(* CODESYS project IndraLogic.project

Project tree, tasks and I/O mapping:
  IndraMotionMlc1 : IndraMotion MLC L75, Bosch Rexroth AG, order no. R911173004, version 14.22.170.0
    application Application
      libraries: SysCallback23, * (System); Util, * (System); RIL_SocketComm, * (System); SysTime23, * (System); SysTaskInfo23, * (System); RIL_CheckRtv, * (System); ML_TechMotion, * (System); SysSocket23, * (System); SysTime, 3.4.1.20 (System); ML_TechInterface, 14.20.30.0 (System); ML_TechBase, 14.18.0.0 (System); VisuDialogs, * (System); ML_TechMotionBase, * (System); RIL_LoopControl, 14.22.36.0 (System); RIL_OpcUaServer, * (System); RIL_OpcUaClient, * (System); IoDrvModbusTCP, * (3S - Smart Software Solutions GmbH)
      task motion (externalevent, external event EVENT_OP_MODE_MOTION_CYCLIC, priority 2) calls P_Position_and_MJD [add POU_1MS below for frequency response tests], P_EL_VEL_MODE, P_PID_antibacklash, P_UDP_To_NTP, POU_20200525, P_Track_cubic, P_Simulation [Just for Simulation PLC remove for pedestal deploy]
      task panel (cyclic, interval t#20ms, priority 7) calls P_remote_local, P_power_on_Sim, P_power_off_TCP
      task TCP (cyclic, interval 10 ms, priority 4) calls P_Opcua_Azimuth [Removed P_TCP_with_SCC], P_Opcua_Elevation, P_Opcua_FeedIndexer, P_Opcua_Safety, P_Opcua_CommandArbiter, P_Opcua_Time_cds, P_Opcua_Management, P_UDP_with_DAM, P_Opcua_Tracking, P_Opcua_Pointing
      task other (cyclic, interval 100 ms, priority 8) calls Test_move, PlcProg
      task AutoStow (cyclic, interval 60000 ms, priority 20) calls P_AutoStow
      function CheckBounds [ST]
      Symbols
      global variables MlcVarGlobal
      POUs/
        Motion/
          program P_PID_antibacklash [ST]: A_PID
          program P_power_off_TCP [LD]
          program P_power_on_TCP [LD]
          program Test_move [ST]: power_move
          program POU_20200525 [ST]
          program PlcProg [ST]
          program P_Position_and_MJD [ST]: A_Write_Limit_Value
          program P_EL_VEL_MODE [ST]
          program P_Track_cubic [ST]: A_track_fuction_blocks, A_StaticPM, A_DynamicPM, A_AmbTempPM, A_Sim_track_function_blocks
          program POU_1MS [ST]: P_Move
          program P_power_on_Sim [LD]
          program P_Read_Parameters [ST]: A_Read_Parameter
          program P_interpolator [ST]: A_track_fuction_blocks, A_StaticPM, A_DynamicPM, A_AmbTempPM, A_Sim_track_function_blocks
        Panel Function/
          program P_LED [ST]: A_w_P304
          program P_Lock_Panel_TCP [ST]: A_LOCK
          program P_Panel_Jog [ST]: A_axes_running
          program P_read_drv_IO [LD]
          program P_remote_local [ST]: A_clear_error
        TCP/
          Message/
            function block FB_add_vector_old_mode [ST]
            function block FB_MSG [ST]
            function block FB_Str_Divide [ST]
            function F_I_number [ST]
            function F_reduce_to_1_bit [ST]
            function F_reduce_to_4_bit [ST]
            function F_RPL [ST]
            function F_RPL_1 [ST]
            function F_RPL_2 [ST]
            function F_Trim [ST]
            function deg2rad [ST]
            function Encoder_to_motor [ST]
            function block FB_add_vector [ST]
            function Encoder_to_motor_old [ST]
            function P_CLOSE_LOOP [ST]
            function block FB_Caculate_position_1 [ST]
            function F_cyclic_position [ST]
            function block CRC16_MODBUS [ST]
          program P_GSTAT_K2STAT [ST]: A_Read_Parameter
          program P_TCP_with_SCC [ST]: Async_TCP, A_RECV, A_SCC_GOTO, A_SCC_POWER, A_SCC_STOP, A_SEND
          program P_UDP_with_DAM [ST]: Async_TCP, A_RECV, A_SEND
        Time Control/
          function F_NTP_Head [ST]
          program P_UDP_To_NTP [ST]: A_NTP_to_Master, A_UDP
        program Annotation [ST]
        Useless/
          program MotionProg [ST]: P_MOTION
          program POU_1MS_Az_freq [ST]
          program POU_1MS_old_mode [ST]: P_Move
        OPCUA/
          OPCUA_Node/
            program P_Opcua_Azimuth [ST]
            program P_Opcua_Elevation [ST]
            program P_Opcua_FeedIndexer [ST]
            program P_Opcua_Safety [ST]: A_STOW, A_Interlock_Estop
            program P_Opcua_CommandArbiter [ST]
            program P_Opcua_Time_cds [ST]: Get_Time
            program P_Opcua_Management [ST]: A_STOP, A_GOTO, A_CLR_ERR
            program P_Opcua_Pointing [ST]: A_Utils
            program P_Opcua_Tracking [ST]: A_Utils
          OPCUA_Method/
            function block fb_Axis [ST]
            function block fb_CommandArbiter [ST]
            function block fb_Management [ST]
            function block fb_Pointing [ST]
            function block fb_Safety [ST]
            function block fb_Time_cds [ST]
            function block fb_Tracking [ST]
            function block fb_Time_Commands [ST]: SetTimeSource
            function block fb_Pointing_Commands [ST]: AmbTempCorrSetup, PmCorrOnOff, StaticPmSetup, TiltCalSetup
            function block fb_Tracking_Commands [ST]: TrackLoadStaticOff, TrackLoadTable, TrackStart, TrackStartPoly
            function block fb_Mngmt_Commands [ST]: Activate, DeActivate, Move2Band, Reset, SetOnSourceThreshold, SetPowerMode, Slew2AbsSingleAx, Slew2AbsAzEl, Slew2RelSingleAx, Slew2RelAzEl, Stop, Stow, TrackStartDM, TrackStartPolyDM
            function block fb_CommandArbiter_Commands [ST]: TakeAuth, ReleaseAuth, Get_Time
            function block fb_Safety_Commands [ST]: InterlockAck, MoveStowPin
        Simulation/
          program P_Simulation [ST]
        AutoStow/
          program P_AutoStow [ST]
      global variables Global_Variables
      Data types/
        data type Stack_buffer
        data type UDP_PACKET
        data type Angle_Mark
        data type ANG_MARK
      global variables UserConstGlobal
      global variables UserVarGlobal
      AxisInterface/
        Documentation/
        Type/
          data type TE_PLC_CYCLES_TIME
          Control/
            data type TE_AXIS_ADMINISTRATION
            data type TE_AXIS_CONTROL_TYPE01
            data type TE_AXIS_POSITIONING
            data type TE_AXIS_SETUP_MODE
            data type TE_AXIS_SYNCHRONISATION
            data type TE_AXIS_TORQUE
            data type TE_AXIS_VELOCITY
          Status/
            data type TE_AXIS_ADMIN_STATUS
            data type TE_AXIS_DATA_STATUS
            data type TE_AXIS_DIAGNOSIS
            data type TE_AXIS_POS_STATUS
            data type TE_AXIS_SETUP_MODE_STATUS
            data type TE_AXIS_STATUS_TYPE01
            data type TE_AXIS_SYNC_STATUS
            data type TE_AXIS_VEL_STATUS
        Visualizations/
          AxisModes/
            text list AxisMode
            text list ExecutionMode
            text list ProfileEntry
            text list StartMode
            text list SyncDirection
            text list SyncType
            visualisation Axis_Overview
            visualisation Position_mode
            visualisation Profile_mode
            visualisation Synchronization_mode
            visualisation Torque_mode
            visualisation Velocity_mode
          ImcInterface/
            text list ImcModeControl
            text list ImcModeStatus
            visualisation ImcControl
            visualisation ImcInterface_Status_Control
            visualisation ImcStatus
          SystemOverview/
            text list ErrorIDCode
            text list ErrorTable
            visualisation System_Overview
            visualisation System_Overview_All_Axis
            visualisation System_Overview_header
          Utilities/
            visualisation AdjustPosition
            visualisation AdjustVelocity
        global variables Global_AxIf_Const
        global variables Global_Axis_Interface
        function block TE_AxisInitAllAxisType01 [ST]
        function block TE_AxisInterface [ST]: actAngleOffset, actCopyAxisData_HMI, actPhaseShift, actPMSpecialErrors, actRetriggerOpMode, actSetupMode, actSyncAccVel, mClearError, mGetOpMode, mInitExtension, mSetOpMode
        program TE_AxisInterfaceType01Prog [ST]: actInitWarmStart
        program _Readme [ST]
      trace/
        trace Trace_simulation (task motion): r_write_position_az, r_write_position_el
        trace Trace_1 (task motion): r_pos_az, r_torque_1, r_torque_2, Global_Variables.i_speed_1, Global_Variables.i_speed_2, i_pos_cmd_1
        trace Trace_2 (task motion, trigger Positive on POU_1MS.r_new_cmd_pos): P_Position_and_MJD.r_test_value, r_following_3, P_Position_and_MJD.b_sign_delay, P_Position_and_MJD.test_1, r_compensation_abs, AxisData[3].rActualTorqueForce_i, r_track_error[2], ML_Base.AxisData[11].rActualPosition_i, r_pos_motor3, P_track_cubic.r_write_position_el, r_vel_EL, P_Track_cubic.r_following_31, P_Position_and_MJD.r_source_to_elevation
        trace Trace_EL_freq_res (task motion): r_pos_motor3, ML_Base.AxisData[11].rActualPosition_i, POU_1MS.Frequency_vel, POU_1MS.vel_freq, POU_1MS.T_period, AxisData[3].rActualVelocity_i, AxisData[3].rActualTorqueForce_i, POU_1MS.torque_freq, Pos_EL_Aim, arAxisCtrl_gb[Drive3.AxisNo].VelMode.Velocity
        trace Trace_compensation (task motion, trigger Positive on POU_1MS.r_new_cmd_pos): r_pos_motor3, ML_Base.AxisData[11].rActualPosition_i, P_Position_and_MJD.test_1, r_track_error[2], AxisData[3].rActualTorqueForce_i, P_Track_cubic.r_write_position_el, P_Track_cubic.r_offset_t, P_Track_cubic.r_test_offset_az, P_Track_cubic.r_test_offset_el
        trace Trace_random_array (task track_task, trigger Positive on POU_1MS.r_new_cmd_pos): ML_Base.AxisData[11].rActualPosition_i, r_pos_motor3, POU_1MS.vel_random_array, AxisData[3].rActualVelocity_i, AxisData[3].rActualTorqueForce_i, POU_1MS.i_test_count, POU_1MS.i_random_count, POU_1MS.vel_freq
        trace Trace_random_array_AZ (task track_task, trigger Positive on POU_1MS.r_new_cmd_pos): ML_Base.AxisData[1].rActualPosition_i, axisdata[1].rActualPosition_i, axisdata[2].rActualPosition_i, POU_1MS.vel_random_array, AxisData[1].rActualVelocity_i, AxisData[1].rActualTorqueForce_i, AxisData[2].rActualTorqueForce_i, POU_1MS.i_test_count, POU_1MS.i_random_count, POU_1MS.vel_random_array
        trace Trace_AZ_freq_res (task motion): ML_Base.AxisData[1].rActualPosition_i, axisdata[1].rActualPosition_i, axisdata[2].rActualPosition_i, POU_1MS.Frequency_vel, AxisData[1].rActualVelocity_i, AxisData[2].rActualVelocity_i, AxisData[1].rActualTorqueForce_i, AxisData[2].rActualTorqueForce_i, POU_1MS.torque_freq, ML_Base.AxisData[11].rActualPosition_i, r_following_1, r_following_3
        trace Trace_EL_VEL_MODE (task motion): r_pos_el, Pos_EL_error, AxisData[3].rActualTorqueForce_i, Pos_EL_Aim, b_step_running, r_vel_EL, AxisData[3].rActualVelocity_i
      global variables PLC_PRG
      OPC_UA_Symbols_Objects/
        data type AxisSelectType
        data type AxisStateType
        data type BandType
        data type CmdResponseType
        data type DscCmdAuthorityType
        data type DscStateType
        data type DscTimeSyncSourceType
        data type InterpolType
        data type LoadModeType
        data type SafetyStateType
        data type StowPinStatusType
        data type TimeSourceType
        data type TiltOnType
      OPCUA_Data_type/
        data type AmbTempParam_Type
        data type AxisErrorStatus_Type
        data type MngmtStatus_Type
        data type MotorStatus_Type
        data type StaticPmParam
        data type TableStatus_type
        data type TiltmeterParam
        data type TiltmeterSubParam
        data type MngmtWarningStatus_Type
        data type SafetyStatus_Type
        data type Time_cdsStatus_type
        data type PointingStatus_Type
        data type TrackingStatus_Type
        data type PolyStatus_type
        data type PowerStatus_Type
        data type AxisWarning_Type
        data type MngmtErrorStatus_Type
        data type TempHumidStatus_Type
        data type NamePlate_Type
        data type CommandArbiter_Status_Type
        data type AxisGeneralStatus_Type
      trace Azimuth_Desired (task TCP, trigger Positive on b_track_on): Tracking.Status.p_desired_Az, Tracking.Status.p_desired_El
    Onboard_I_O : Onboard I/O, Bosch Rexroth AG, version 13.6.2.0
        unmapped channels: OnboardIn, OnboardOut
    Inline_I_O : Inline I/O, Bosch Rexroth AG, version 12.8.2.0
      R_IB_IL_24_DI_32_HD : R-IB IL 24 DI 32/HD, Bosch Rexroth AG, order no. R911170753, R911297188, version 0.0.0.1
          unmapped channels: Input0
      R_IB_IL_24_DO_32_HD : R-IB IL 24 DO 32/HD, Bosch Rexroth AG, order no. R911170411, R911297191, version 0.0.0.1
          unmapped channels: Output0
    Not_Used : Not Used, Bosch Rexroth AG, version 12.2.0.0
    EtherNet_IP_Adapter : EtherNet/IP Adapter, Bosch Rexroth AG, version 14.22.10.0
    Sercos_III_Master : SercosIII Master, Rexroth, order no. 1, version 14.6.0.0
    EtherNet_IP_Adapter_on_Eng_Port : EtherNet/IP Adapter on Eng.-Port, Bosch Rexroth AG, version 12.10.2.0
      _8_Byte_Input : 8 Byte Input, Bosch Rexroth AG, version 12.10.2.0
          unmapped channels: Channel1
      _8_Byte_Output_4Byte_Run_Header : 8 Byte Output + 4Byte Run Header, Bosch Rexroth AG, version 12.10.2.0
          unmapped channels: Channel1
  libraries: Time and Date, 3.5.7.0 (3S - Smart Software Solutions GmbH); Util, * (System); RIL_OpcUaServer, 14.22.0.1 (System); RIL_LoopControl, 14.22.36.0 (System); RIL_EtherNetIPAdapter, 14.4.0.0 (System); ML_PLCopen, 14.22.32.0 (System); IoDrvModbusTCP, * (3S - Smart Software Solutions GmbH)
  text list GlobalTextList
  visualisation Visualization
*)

// IndraMotionMlc1/Application/OPCUA_Data_type/AmbTempParam_Type
TYPE AmbTempParam_Type :
STRUCT
	AmbTempParam1:LREAL;
	AmbTempParam2:LREAL;
	AmbTempParam3:LREAL;
	AmbTempParam4:LREAL;
	AmbTempParam5:LREAL;
	AmbTempParam6:LREAL;
	Filt_dt:LREAL;
END_STRUCT
END_TYPE

// IndraMotionMlc1/Application/Data types/Stack_buffer
(*construction of stack *)
TYPE Stack_buffer :
STRUCT
	TAIoffset:LREAL;
	Azimuth:LREAL;
	Elevation:LREAL;
	//FeedIndexer:LREAL;
	//Elevation_ori:LREAL;
END_STRUCT
END_TYPE

// IndraMotionMlc1/Application/Data types/UDP_PACKET
TYPE UDP_PACKET :(*constrution of NTP header*)
STRUCT
	(*NTP packet = NTP header 16bytes + Four TimeStamps 32 byte = 48byte*)
	NTP_Header :ARRAY[1..4] OF BYTE;
	NTP_Root_Delay:ARRAY[1..4] OF BYTE;
	NTP_Root_Dispersion:ARRAY[1..4] OF BYTE;
	NTP_Reference_Identifier:ARRAY[1..4] OF BYTE;

	NTP_Reference_Timestamp:ARRAY[1..2] OF DWORD;
	NTP_Originate_Timestamp:ARRAY[1..2] OF DWORD;
	NTP_Receive_Timestamp:ARRAY[1..2] OF DWORD;
	NTP_Transmit_Timestamp:ARRAY[1..2] OF DWORD;
END_STRUCT
END_TYPE

// IndraMotionMlc1/Application/Data types/Angle_Mark
TYPE Angle_Mark :
STRUCT
	stui_RSV : DINT;			//补齐8字节，对齐地址
	stui_SID : DINT;
	stui_DID : DINT;
	stui_BID : DINT;
	stui_DataLen : DINT;
	sti_Year : DINT;
	sti_Month : DINT;
	sti_Day : DINT;
	sti_Hour : DINT;
	sti_Minute : DINT;
	sti_Second : DINT;
	sti_MilSecond : DINT;
	std_GEOAngle_AZ : LREAL;
	std_GEOAngle_EL : LREAL;
END_STRUCT
END_TYPE

// IndraMotionMlc1/Application/Data types/ANG_MARK
TYPE ANG_MARK :
UNION
	st_ANGMARK : Angle_Mark;
	ANG_SEND : ARRAY [1..64] OF BYTE;
END_UNION
END_TYPE

// IndraMotionMlc1/Application/AxisInterface/Type/TE_PLC_CYCLES_TIME
TYPE TE_PLC_CYCLES_TIME :
STRUCT

     udiMinimumTime  : UDINT  := 1000000;
     udiActualTime   : UDINT  := 0;
     udiMaximumTime  : UDINT  := 0;

END_STRUCT
END_TYPE

// IndraMotionMlc1/Application/AxisInterface/Type/Control/TE_AXIS_ADMINISTRATION
// Online changes in declaration of axis-interface need too much time -> not allowed because risk of F5180006 
// InhibitOnlineChange = 0x1000000 has to be set decimal 16777216
{attribute 'signature_flag' := '16777216'} 
TYPE TE_AXIS_ADMINISTRATION EXTENDS MB_AXIS_ADMINISTRATION:
STRUCT
  (* add your extensions below here |  Erweiterungen hier einfuegen*)

  (* user extensions | Anwender Erweiterungen *)
  
  RetriggerOpMode: BOOL;   // Restart the same OpMode again, e.g. MoveRelative with same distance	

END_STRUCT
END_TYPE

// IndraMotionMlc1/Application/AxisInterface/Type/Control/TE_AXIS_CONTROL_TYPE01
// Online changes in declaration of axis-interface need too much time -> not allowed because risk of F5180006 
// InhibitOnlineChange = 0x1000000 has to be set decimal 16777216
{attribute 'signature_flag' := '16777216'} 
TYPE TE_AXIS_CONTROL_TYPE01:

STRUCT
    Admin:      TE_AXIS_ADMINISTRATION; (* Administration of the axis | Verwaltung der Achse *)

    PosMode:    TE_AXIS_POSITIONING; (* operating mode positioning (absolute, rel. and additive)
      Positionierbetrieb (absolut, relativ und additiv) *)

    VelMode:    TE_AXIS_VELOCITY; (* operating mode velocity control | Geschwindigkeitsregelung *)

    SyncMode:   TE_AXIS_SYNCHRONISATION; (* operating mode synchronisation (phase, vel, and cam)
      Synchronbetriebsarten (Winkelsync., Geschwindigkeitssync. und Kurvenscheibe) *)
			
    TorqueMode: TE_AXIS_TORQUE; (* operating mode torque/force control | Drehmoment-/Kraftregelung *)

    (* add your extensions below here, keep the elements above
       Erweiterungen hier einfuegen, Elemente oberhalb nicht veraendern *)

    (* user extensions | Anwender Erweiterungen *)
    
	  // Jog/Homing functionality | Tipp/Einrichtfunktionen 
    SetupMode:  TE_AXIS_SETUP_MODE; 
	
END_STRUCT

END_TYPE

// IndraMotionMlc1/Application/AxisInterface/Type/Control/TE_AXIS_POSITIONING
    (*************** - setpoints of positioning mode ******************)
    (*************** - Positions-Sollwerte           ******************)
// Online changes in declaration of axis-interface need too much time -> not allowed because risk of F5180006 
// InhibitOnlineChange = 0x1000000 has to be set decimal 16777216
{attribute 'signature_flag' := '16777216'} 
TYPE TE_AXIS_POSITIONING EXTENDS MB_AXIS_POSITIONING:
STRUCT

    (* position for an absolute move (in technical unit[u]) (negative or positive)
      - start moving with "ModePosAbs" (MC_MoveAbsolute)
      Note: cyclic checked AND transmitted on change (EnableCyclicScanning = TRUE) 
      ------------------------------------------------------------------------------
      Zielposition, absolut (Einheit: [u]) (negativ oder positiv)
      - Freigabe mit "ModePosAbs" (MC_MoveAbsolute)
      Hinweis: wird permanent zyklisch verarbeitet (EnableCyclicScanning = TRUE) *)
    // Position:        REAL;

    (* distance for a relative or additive move (in technical unit[u]) (negative or positive)
      - start moving with "ModePosRel" or "ModePosAdd" (MC_MoveRelative, MC_MoveAdditive) 
      Note: cyclic checked AND transmitted on change (EnableCyclicScanning = TRUE) 
      ------------------------------------------------------------------------------
      Relativer / additiver Sollwert (Einheit: [u]) (negativ oder positiv )
      - Freigabe mit "ModePosRel" oder "ModePosAdd" (MC_MoveRelative, MC_MoveAdditive) 
      Hinweis: wird permanent zyklisch verarbeitet (EnableCyclicScanning = TRUE) *)
     // Distance:        REAL;

    (* maximum velocity (always positive) (not necessarily reached) [u/s]
      - start moving with "ModePosAbs" or "ModePosRel" or "ModePosAdd" 
        (MC_MoveAbsolute, MC_MoveRelative, MC_MoveAdditive) 
      Note: cyclic checked AND transmitted on change (EnableCyclicScanning = TRUE) 
      ------------------------------------------------------------------------------
      Positioniergeschwindigkeit , (Einheit: [u/s]) (positiv eingeben)
      - Freigabe mit "ModePosAbs" oder "ModePosRel" oder "ModePosAdd" 
        (MC_MoveAbsolute, MC_MoveRelative, MC_MoveAdditive) 
      Hinweis: wird permanent zyklisch verarbeitet (EnableCyclicScanning = TRUE) *)
    // Velocity:        REAL:=10.0;

    (* Value of the acceleration (always positive) (increasing energy of the motor) [u/s2]
      - start moving with "ModePosAbs" or "ModePosRel" or "ModePosAdd" 
        (MC_MoveAbsolute, MC_MoveRelative, MC_MoveAdditive) 
      ------------------------------------------------------------------------------
      Beschleunigung (Einheit: [u/s2]) (nur positive Werte)             
      - Freigabe mit "ModePosAbs" oder "ModePosRel" oder "ModePosAdd" 
        (MC_MoveAbsolute, MC_MoveRelative, MC_MoveAdditive) *)
    // Acceleration:    REAL:=10.0;

    (* Value of the deceleration (always positive) (decreasing energy of the motor) [u/s2]
      - start moving with ModePosAbs or ModePosRel or ModePosAdd 
        (MC_MoveAbsolute, MC_MoveRelative, MC_MoveAdditive) 
      ------------------------------------------------------------------------------
      Verzoegerung, (Einheit: [u/s2]) (nur positive Werte)            
      - Freigabe mit "ModePosAbs" oder "ModePosRel" oder "ModePosAdd" 
        (MC_MoveAbsolute, MC_MoveRelative, MC_MoveAdditive) *)
    // Deceleration:    REAL:=10.0;
	
(* add your extensions below here, keep the elements above
   Erweiterungen hier einfuegen, Elemente oberhalb nicht veraendern *)

(* user extensions | Anwender Erweiterungen *)

END_STRUCT
END_TYPE

// IndraMotionMlc1/Application/AxisInterface/Type/Control/TE_AXIS_SETUP_MODE
// Online changes in declaration of axis-interface need too much time -> not allowed because risk of F5180006 
// InhibitOnlineChange = 0x1000000 has to be set decimal 16777216
{attribute 'signature_flag' := '16777216'} 
TYPE TE_AXIS_SETUP_MODE :
  STRUCT
    Enable:          BOOL;	  (* Enable setup mode  | Freigabe Einrichtbetrieb
      - activates Power                        | - aktiviert Antriebsfreigabe *)
 
    JogPlus:         BOOL;  	(* Jog +            | Tippen + 
      - activates ModeVelocity with pos. Vel   | - aktiviert ModeVelocity mit pos. Vel *)
 
    JogMinus:        BOOL;    (* Jog -            | Tippen - 
      - activates ModeVelocity with pos. Vel   | - aktiviert ModeVelocity mit neg. Vel *)

    JogPosControl:   BOOL:=FALSE; (* Select jog in velocity or positioning control | Auswahl tippen in Geschwindigkeits- oder Lageregelung 
           TRUE = jog in positioning control | TRUE = tippen in Lageregelung *)

	  (* Homing *)
    {attribute 'analysis' := '-27'} // disable static code analysis rule 27, check of same names 
    Homing: BOOL;  (* - activates ModeHoming|SetAbsRef|ModesPosAbs | activiert ModeHoming|SetAbsRef|ModesPosAbs
        depending on axistype/-configuration       | abhängig vom Achstyp/-konfiguration       *) 

	
    Vel:    REAL:= 10; (* jog/homing velocity  | Tipp-/Referenzfahrgeschwindigkeit *)
	
    Accel:  REAL:= 10; (* jog/homing ac/deceleration  | Tipp/Referenzfahr (brems)beschleunigung *)
  END_STRUCT
END_TYPE

// IndraMotionMlc1/Application/AxisInterface/Type/Control/TE_AXIS_SYNCHRONISATION
    (*************** - setpoint of synchronous motion ******************)
// Online changes in declaration of axis-interface need too much time -> not allowed because risk of F5180006 
// InhibitOnlineChange = 0x1000000 has to be set decimal 16777216
{attribute 'signature_flag' := '16777216'} 
TYPE TE_AXIS_SYNCHRONISATION EXTENDS MB_AXIS_SYNCHRONISATION:
STRUCT

    (* Electronic gear input revolution
      - "ModeSyncPhase", "ModeSyncVel", "ModeSyncCam", "ModeSyncProfile", "ModeFlexProfile"
      - RatioNumerator for MC_GearIn, MB_GearInPos, MC_CamIn, MB_MotionProfile, ML_FlexProfile 
      Note: cyclic checked AND transmitted on change (EnableCyclicScanning = TRUE) 
      ------------------------------------------------------------------------------
      Elektronisches Getriebe, Eingangsumdrehungen
      - "ModeSyncPhase", "ModeSyncVel", "ModeSyncCam", "ModeSyncProfile", "ModeFlexProfile"
      - RatioNumerator fuer MC_GearIn, MB_GearInPos, MC_CamIn, MB_MotionProfile, ML_FlexProfile 
      Hinweis: wird permanent zyklisch verarbeitet (EnableCyclicScanning = TRUE) *)
    // InputRevolution: UINT:=1;

    (* Electronic gear output revolution
      - "ModeSyncPhase", "ModeSyncVel", "ModeSyncCam", "ModeSyncProfile", "ModeFlexProfile"
      - RatioDenominator for MC_GearIn, MB_GearInPos, MC_CamIn, MB_MotionProfile, ML_FlexProfile 
      Note: cyclic checked AND transmitted on change (EnableCyclicScanning = TRUE)
      ------------------------------------------------------------------------------
      Elektronisches Getriebe, Ausgangsumdrehungen
      - "ModeSyncPhase", "ModeSyncVel", "ModeSyncCam", "ModeSyncProfile", "ModeFlexProfile"
      - RatioDenominator fuer MC_GearIn, MB_GearInPos, MC_CamIn, MB_MotionProfile, ML_FlexProfile 
      Hinweis: wird permanent zyklisch verarbeitet (EnableCyclicScanning = TRUE) *)
    // OutputRevolution: UINT:=1;

    (* Master fine adjust
      - "ModeSyncPhase", "ModeSyncVel", "ModeSyncCam", "ModeSyncProfile", "ModeFlexProfile"
      - MasterFineadjust for MC_GearIn, MB_GearInPos, MC_CamIn, MB_MotionProfile, ML_FlexProfile
      Note: cyclic checked AND transmitted on change (EnableCyclicScanning = TRUE) 
      ------------------------------------------------------------------------------
      Getriebe-Feinabgleich
      - "ModeSyncPhase", "ModeSyncVel", "ModeSyncCam", "ModeSyncProfile", "ModeFlexProfile"
      - MasterFineadjust fuer MC_GearIn, MB_GearInPos, MC_CamIn, MB_MotionProfile, ML_FlexProfile
      Hinweis: wird permanent zyklisch verarbeitet (EnableCyclicScanning = TRUE) *)
    // FineAdjust:    REAL:=0.0;

    (* Cam Shaft Distance
      - start moving with "ModeSyncCam"
      - CamShaftDist for MC_CamIn
      Note: cyclic checked AND transmitted on change (EnableCyclicScanning = TRUE) 
      ------------------------------------------------------------------------------
      Kurvenscheibe, Hub
      - Freigabe mit "ModeSyncCam" 
      - CamShaftDist fuer MC_CamIn
      Hinweis: wird permanent zyklisch verarbeitet (EnableCyclicScanning = TRUE) *)
    // CamShaftDistance: REAL:=360.0;

    (* Phase offset between master and slave axis
      - "ModeSyncPhase", "ModeSyncCam", "ModeSyncProfile", "ModeFlexProfile" 
      - PhaseShift for MB_PhasingSlave
      Note: cyclic checked AND transmitted on change (EnableCyclicScanning = TRUE) 
      ------------------------------------------------------------------------------
      Winkelversatz (Lagesollwert additiv)
      - "ModeSyncPhase", "ModeSyncCam", "ModeSyncProfile", "ModeFlexProfile" 
      - PhaseShift fuer MB_PhasingSlave
      Hinweis: wird permanent zyklisch verarbeitet (EnableCyclicScanning = TRUE) *)
    // PhaseOffset:   REAL:=0.0; 

    (* Velocity for the phase offset
      - "ModeSyncPhase", "ModeSyncCam", "ModeSyncProfile", "ModeFlexProfile"
      - Velocity for MB_PhasingSlave 
      ------------------------------------------------------------------------------
      Aufsynchronisier-Geschwindigkeit
      - "ModeSyncPhase", "ModeSyncCam", "ModeSyncProfile", "ModeFlexProfile"
      - Velocity fuer MB_PhasingSlave *)
	// PhaseOffsetVel: REAL:=1.0;

    (* Acceleration for the phase offset
      - "ModeSyncPhase", "ModeSyncCam", "ModeSyncProfile", "ModeFlexProfile" 
      - PhaseShift for MB_PhasingSlave
      ------------------------------------------------------------------------------
      Aufsynchronisier-Beschleunigung
      - Freigabe mit "ModeSyncPhase", "ModeSyncCam" oder "ModeSyncProfile"
      - PhaseShift fuer MB_PhasingSlave *)
    // PhaseOffsetAcc: REAL:=100.0;

    (* Synchronisation direction
      - values 'SHORTEST_WAY'; 'CATCH_UP' (always forward); 'SLOW_DOWN' (see RIL_CommonTypes.lib)
      - start moving with "ModeSyncPhase", "ModeSyncCam" or "ModeSyncProfile"
      - SyncMode for MB_GearInPos, MC_CamIn, MB_MotionProfile 
      ------------------------------------------------------------------------------
      Aufsynchronisier-Richtung
      - Werte 'SHORTEST_WAY'; 'CATCH_UP' (positiv); 'SLOW_DOWN' (siehe RIL_CommonTypes.lib)
      - Freigabe mit "ModeSyncPhase", "ModeSyncCam" oder "ModeSyncProfile"
      - SyncMode fuer MB_GearInPos, MC_CamIn, MB_MotionProfile *)
    // SyncDirection: MC_SYNC_DIRECTION:= SHORTEST_WAY;

    (* Start mode of the synchronisation
      - values 'ABSOLUTE'; 'RELATIVE' (see RIL_CommonTypes.lib)
      - start moving with "ModeSyncPhase", "ModeSyncCam" or "ModeSyncProfile"
      - StartMode for MB_GearInPos, MC_CamIn, MB_MotionProfile 
      ------------------------------------------------------------------------------
      Aufsynchronisier-Mode
      - Werte: 'ABSOLUTE'; 'RELATIVE' (siehe RIL_CommonTypes.lib)
      - Freigabe mit "ModeSyncPhase", "ModeSyncCam" oder "ModeSyncProfile"
      - StartMode fuer MB_GearInPos, MC_CamIn, MB_MotionProfile *)
    // StartMode:     MC_START_MODE:= ABSOLUTE;

    (* Number of the selected cam table
      - values 'CAM_TABLE_1'; 'CAM_TABLE_2' ... 'CAM_TABLE_8' (see RIL_CommonTypes.lib)
      - start moving with "ModeSyncCam" 
      - CamTableID for MC_CamIn
      Note: cyclic checked AND transmitted on change (EnableCyclicScanning = TRUE)
      ------------------------------------------------------------------------------
      Nummer Stuetzpunkt-Tabelle
      - Werte: 'CAM_TABLE_1'; 'CAM_TABLE_2' ... 'CAM_TABLE_8' (siehe RIL_CommonTypes.lib)
      - Freigabe mit "ModeSyncCam" 
      - CamTableID fuer MC_CamIn
      Hinweis: wird permanent zyklisch verarbeitet (EnableCyclicScanning = TRUE) *)
    // CamTableID:    MC_CAM_ID:= CAM_TABLE_1;

    (* -> AXIS_REF of the master axis
      - "ModeSyncPhase", "ModeSyncVel", "ModeSyncCam", "ModeSyncProfile", "ModeFlexProfile"
      - Master for MC_GearIn, MB_GearInPos, MC_CamIn, MB_MotionProfile, ML_FlexProfile 
      Note: cyclic checked AND transmitted on change (EnableCyclicScanning = TRUE)
      ------------------------------------------------------------------------------
      -> AXIS_REF der Leitachse
      - "ModeSyncPhase", "ModeSyncVel", "ModeSyncCam", "ModeSyncProfile", "ModeFlexProfile"
      - Master fuer MC_GearIn, MB_GearInPos, MC_CamIn, MB_MotionProfile, ML_FlexProfile 
         Hinweis: wird permanent zyklisch verarbeitet (EnableCyclicScanning = TRUE) *)
    // Master:    AXIS_REF    := (AxisNo := NO_OBJECT, CntrlNo := LOCAL_CNTRL);


    (*************** Extensions for profile operation modes *******************)
    (************* Erweiterungen für die Profil Betriebsarten *****************)
    (* Extensions for the operating modes MotionProfile and FlexProfile
       ------------------------------------------------------------------------------
       Erweiterungen füt die Betriebsarten MotionProfile und FlexProfile *)
    // Profile:     ML_AXIS_PROFILE;
	
  (* add your extensions below here, keep the elements above
     Erweiterungen hier einfuegen, Elemente oberhalb nicht veraendern *)

  (* user extensions | Anwender Erweiterungen *)

	AngleOffset:   REAL:= 0;   // angle offset begin of profile | Winkelverschiebung Tabellenanfang  
	
  // Values for MB_Phasing | Werte für MB_Phasing
	PhaseShift:    REAL:=0.0;    // Additive master position command value (MB_Phasing)    
	PhaseShiftVel: REAL:=10.0;   // Additive master position velocity (MB_Phasing) 
	PhaseShiftAcc: REAL:=100.0;  // Additive master position acceleration (MB_Phasing)
  
  SyncVelocity:     REAL := 10.0;   // A-0-2790 Synchronisation velocity | Aufsynchronisiergeschw. 

  SyncAcceleration: REAL := 10.0;   // A-0-2791 Synchron. acceleration | Aufsynchronisierbeschleunigung 

END_STRUCT
END_TYPE

// IndraMotionMlc1/Application/AxisInterface/Type/Control/TE_AXIS_TORQUE
    (*************** - setpoints of velocity mode                    ************)
    (*************** - Sollwerte Geschwindigkeitsregelung (Freilauf) ************)
// Online changes in declaration of axis-interface need too much time -> not allowed because risk of F5180006 
// InhibitOnlineChange = 0x1000000 has to be set decimal 16777216
{attribute 'signature_flag' := '16777216'} 
TYPE TE_AXIS_TORQUE EXTENDS MB_AXIS_TORQUE:
STRUCT

    (*Maximum value of the power/torque (Unit: e.g. in [%] or [Nm] depending on 
      parametrization) 
      Value always positive, value does not necessarily have to be reached 
      - start moving with "ModeTorque" (MC_TorqueControl)
      Note: cyclic checked AND transmitted on change (EnableCyclicScanning = TRUE) 
      -----------------------------------------------------------------------------
      Maximalwert der Kraft/ des Drehmomentes (Einheit: z.B. in in [%] oder [Nm] 
      je nach Parametrierung)
      Wert stets positiv, Wert muss nicht unbedingt erreicht werden 
      - Freigabe mit "ModeTorque" (MC_TorqueControl)
      Hinweis: wird permanent zyklisch verarbeitet (EnableCyclicScanning = TRUE) *)
    //Torque:        REAL:=0.0;

    (*Power/torque difference which can be reached within the ramp time
      Unit: e.g. in [%/s] or [Nm/s] depending on parametrization (always positive)
      - start moving with "ModeTorque" (MC_TorqueControl)
      Note: cyclic checked AND transmitted on change (EnableCyclicScanning = TRUE) 
      -----------------------------------------------------------------------------
			Kraft-/ Drehmoment-Differenz, die innerhalb der Rampenzeit erreicht werden kann
      Einheit: z.B. in [%/s] oder [Nm/s] je nach Parametrierung (immer positiv)       
      - Freigabe mit "ModeTorque" (MC_TorqueControl)
      Hinweis: wird permanent zyklisch verarbeitet (EnableCyclicScanning = TRUE) *)
    //TorqueRamp:    REAL:=10.0;

(* add your extensions below here, keep the elements above
   Erweiterungen hier einfuegen, Elemente oberhalb nicht veraendern *)

(* user extensions | Anwender Erweiterungen *)

END_STRUCT
END_TYPE

// IndraMotionMlc1/Application/AxisInterface/Type/Control/TE_AXIS_VELOCITY
    (*************** - setpoints of velocity mode                    ************)
    (*************** - Sollwerte Geschwindigkeitsregelung (Freilauf) ************)
// Online changes in declaration of axis-interface need too much time -> not allowed because risk of F5180006 
// InhibitOnlineChange = 0x1000000 has to be set decimal 16777216
{attribute 'signature_flag' := '16777216'} 
TYPE TE_AXIS_VELOCITY EXTENDS MB_AXIS_VELOCITY:
STRUCT

    (* Value of the maximum velocity (Unit: [u/s])
      - start moving with "ModeVel" (MC_MoveVelocity)
      Note: cyclic checked AND transmitted on change (EnableCyclicScanning = TRUE) 
      -----------------------------------------------------------------------------
      Geschwindigkeits-Sollwert, (Einheit: [u/s]) 
      - Freigabe mit "ModeVel" (MC_MoveVelocity)
      Hinweis: wird permanent zyklisch verarbeitet (EnableCyclicScanning = TRUE) *)
    // Velocity:        REAL:=0.0;

    (* Value of the acceleration and deceleration [u/s2] (always positive)
      - start moving with "ModeVel" (MC_MoveVelocity)
      -----------------------------------------------------------------------------
      Beschleunigung, (Einheit: [u/s2]) (immer positiv eingeben)            
      - Freigabe mit "ModeVel" (MC_MoveVelocity) *)
    // Acceleration:    REAL:=10.0;

    (* Value of the deceleration [u/s2] (always positive)
      - start moving with "ModeVel" (MC_MoveVelocity) 
      -----------------------------------------------------------------------------
      Verzoegerung, (Einheit: [u/s2]) (immer positiv eingeben)
      - Freigabe mit "ModeVel" (MC_MoveVelocity) *)
    // Deceleration:    REAL:=10.0;
	
(* add your extensions below here, keep the elements above
   Erweiterungen hier einfuegen, Elemente oberhalb nicht veraendern *)

(* user extensions | Anwender Erweiterungen *)

END_STRUCT
END_TYPE

// IndraMotionMlc1/Application/AxisInterface/Type/Status/TE_AXIS_ADMIN_STATUS
    (********** Administrative outputs - from motion control to logic control *****************)
    (********** Administrative Ausgaenge - Motion Control zur Logic Control   *****************)
// Online changes in declaration of axis-interface need too much time -> not allowed because risk of F5180006 
// InhibitOnlineChange = 0x1000000 has to be set decimal 16777216
{attribute 'signature_flag' := '16777216'} 
TYPE TE_AXIS_ADMIN_STATUS EXTENDS MB_AXIS_ADMIN_STATUS:

STRUCT
  (* add your extensions below here |  Erweiterungen hier einfuegen*)

  (* User extensions | Anwender Erweiterungen *)

 
END_STRUCT

END_TYPE

// IndraMotionMlc1/Application/AxisInterface/Type/Status/TE_AXIS_DATA_STATUS
// Online changes in declaration of axis-interface need too much time -> not allowed because risk of F5180006 
// InhibitOnlineChange = 0x1000000 has to be set decimal 16777216
{attribute 'signature_flag' := '16777216'} 
TYPE TE_AXIS_DATA_STATUS :
STRUCT
	                  dwMotionProfileStatusBits_i     :DWORD;      (* A-0-2931 -RD- Motion profile status word *)
                      FlexProfil_Sync                 :BOOL;       (* A-0-3010.08 -RD- FlexProfile is in synchronisation *)
                      FlexProfil_Active               :BOOL;       (* A-0-3010.09 -RD- FlexProfile is active *)
                      FlexProfil_WaitForSwitching     :BOOL;       (* A-0-3010.10 -RD- FlexProfile is waiting for switching position *)
                      FlexProfil_Set0_Checked         :BOOL;       (* A-0-3010.16 -RD- FlexProfile Set0 is checked *)
                      FlexProfil_Set0_Ok              :BOOL;       (* A-0-3010.17 -RD- FlexProfile Set0 is ok *)
                      FlexProfil_Set1_Checked         :BOOL;       (* A-0-3010.18 -RD- FlexProfile Set0 is checked *)
                      FlexProfil_Set1_Ok              :BOOL;       (* A-0-3010.19 -RD- FlexProfile Set0 is ok *)
                      FlexProfil_Set2_Checked         :BOOL;       (* A-0-3010.20 -RD- FlexProfile Set0 is checked *)
                      FlexProfil_Set2_Ok              :BOOL;       (* A-0-3010.21 -RD- FlexProfile Set0 is ok *)
                      FlexProfil_Set3_Checked         :BOOL;       (* A-0-3010.22 -RD- FlexProfile Set0 is checked *)
                      FlexProfil_Set3_Ok              :BOOL;       (* A-0-3010.23 -RD- FlexProfile Set0 is ok *)
                      FlexProfil_EvtSet0_Checked      :BOOL;       (* A-0-3010.24 -RD- FlexProfile Event Set0 is checked *)
                      FlexProfil_EvtSet0_Ok           :BOOL;       (* A-0-3010.25 -RD- FlexProfile Event Set0 is ok *)
                      FlexProfil_EvtSet1_Checked      :BOOL;       (* A-0-3010.26 -RD- FlexProfile Event Set0 is checked *)
                      FlexProfil_EvtSet1_Ok           :BOOL;       (* A-0-3010.27 -RD- FlexProfile Event Set0 is ok *)
                      FlexProfil_EvtSet2_Checked      :BOOL;       (* A-0-3010.28 -RD- FlexProfile Event Set0 is checked *)
                      FlexProfil_EvtSet2_Ok           :BOOL;       (* A-0-3010.29 -RD- FlexProfile Event Set0 is ok *)
                      FlexProfil_EvtSet3_Checked      :BOOL;       (* A-0-3010.30 -RD- FlexProfile Event Set0 is checked *)
                      FlexProfil_EvtSet3_Ok           :BOOL;       (* A-0-3010.31 -RD- FlexProfile Event Set0 is ok *)
                      dwFlexProfileEventStatusBits_i  :DWORD;      (* A-0-3012 -RD- Condition status variable, FlexProfile *)

                      Axis_CamTab_0                   :BOOL;       (* A-0-0021.00 -RD- Cam shaft table BOOL 0 *)                
                      Axis_CamTab_1                   :BOOL;       (* A-0-0021.01 -RD- Cam shaft table BOOL 1 *)
                      Axis_CamTab_2                   :BOOL;       (* A-0-0021.02 -RD- Cam shaft table BOOL 2 (reserved) *)
                      Axis_CamSwitching               :BOOL;       (* A-0-0021.03 -RD- Status cam shaft distance switching *)
                      Axis_InVelocity                 :BOOL;       (* A-0-0021.04 -RD- Axis cmd velocity == actual velocity *)
                      Axis_Standstill                 :BOOL;       (* A-0-0021.05 -RD- Axis velocity <= A-0-0222 (standstill) *)
                      Axis_InPosition                 :BOOL;       (* A-0-0021.06 -RD- Axis cmd position == actual position *)
                      Axis_InSynchron                 :BOOL;       (* A-0-0021.07 -RD- Axis is in synchronisation *)
                      Axis_Warning                    :BOOL;       (* A-0-0021.08 -RD- Axis reports warning *)
                      Axis_Error                      :BOOL;       (* A-0-0021.09 -RD- Axis reports error *)
                      Axis_Homed                      :BOOL;       (* A-0-0021.10 -RD- Axis is relative / in homing *)
                      Axis_InTorque                   :BOOL;       (* A-0-0021.11 -RD- Axis cmd torque / force == actual torque *)
                      Axis_OperationMode              :BOOL;       (* A-0-0021.12 -RD- Axis is in operation mode (P4) *)
                      Axis_Inbb                       :BOOL;       (* A-0-0021.13 -RD- Axis is ready for power to the amplifier (bb) *)
                      Axis_InAb                       :BOOL;       (* A-0-0021.14 -RD- Axis is ready for power to the engine (Ab) *)
                      Axis_Power                      :BOOL;       (* A-0-0021.15 -RD- Axis has power on (AH_AF) *)
                      Axis_CmdActive                  :BOOL;       (* A-0-0021.16 -RD- Command active *)
                      Axis_ErrInProgress              :BOOL;       (* A-0-0021.17 -RD- Error reaction in progress *)
                      Axis_CyclicPosChannelOpen       :BOOL;       (* A-0-0021.18 -RD- Cyclic Position Channel is open for Axis *)          
                      Axis_InMasterPhaseOffset        :BOOL;       (* A-0-0021.19 -RD- Master Phase offset achieved *)
                      Axis_CyclicTrqChannelOpen       :BOOL;       (* A-0-0021.20 -RD- Cyclic Position Channel is open for Axis *)          
                      Axis_CyclicVelChannelOpen       :BOOL;       (* A-0-0021.21 -RD- Cyclic Position Channel is open for Axis *)          
                      Axis_CyclicAnaChannelOpen       :BOOL;       (* A-0-0021.22 -RD- Cyclic Position Channel is open for Axis *)          
                      {attribute 'analysis' := '-27'} // disable static code analysis rule 27, check of same names 
                      ErrorStop                       :BOOL;       (* A-0-0022.00 -RD- Axis is in "ErrorStop" *)
                      {attribute 'analysis' := '-27'} // disable static code analysis rule 27, check of same names 
                      Stopping                        :BOOL;       (* A-0-0022.01 -RD- Axis is in "Stopping" *)
                      {attribute 'analysis' := '-27'} // disable static code analysis rule 27, check of same names 
                      Homing                          :BOOL;       (* A-0-0022.02 -RD- Command homing is active *)
                      {attribute 'analysis' := '-27'} // disable static code analysis rule 27, check of same names 
                      PowerOn                         :BOOL;       (* A-0-0022.03 -RD- Axis got power *)
                      {attribute 'analysis' := '-27'} // disable static code analysis rule 27, check of same names 
                      DiscreteMotion                  :BOOL;       (* A-0-0022.04 -RD- Axis is in "Discrete Motion" *)
                      {attribute 'analysis' := '-27'} // disable static code analysis rule 27, check of same names 
                      ContinuousMotion                :BOOL;       (* A-0-0022.05 -RD- Axis is in "Continuous Motion" *)
                      {attribute 'analysis' := '-27'} // disable static code analysis rule 27, check of same names 
                      SynchronizedMotion              :BOOL;       (* A-0-0022.06 -RD- Axis is in "Synchronized Motion" *)
                      {attribute 'analysis' := '-27'} // disable static code analysis rule 27, check of same names 
                      Standstill                      :BOOL;       (* A-0-0022.07 -RD- Axis is stopped *)
                      CoordinatedMotion               :BOOL;       (* A-0-0022.08 -RD- Axis is in "CoordinatedMotion" *)
                      ControlledMotion                :BOOL;       (* A-0-0022.09 -RD- Axis is in "ControlledMotion" *)  
                      dwAxisCondition_i               :DWORD;      (* A-0-0024 -RD- Axis condition *)
                      rActualPosition_i               :REAL;       (* A-0-0100 -RD- Actual position *)
                      rActualVelocity_i               :REAL;       (* A-0-0102 -RD- Actual velocity *)
                      rActualTorqueForce_i            :REAL;       (* A-0-0110 -RD- Actual torque/force *)
                                                                                 
                    
                      wUserActualDataBitA_i           :WORD;      (* A-0-0562 -RD- User defined actual data BOOL number A, Type: WORD *)
                      wUserActualDataBitB_i           :WORD;      (* A-0-0565 -RD- User defined actual data BOOL number B, Type: WORD *)
                      wUserActualDataBitC_i           :WORD;      (* A-0-0568 -RD- User defined actual data BOOL number C, Type: WORD *)
                      wUserActualDataBitD_i           :WORD;      (* A-0-0571 -RD- User defined actual data BOOL number D, Type: WORD *)
                    
                      dwUserActualDataA_i             :SM_TYPES;  (* A-0-0521 -RD- Container user defined actual data A *)
                      dwUserActualDataB_i             :SM_TYPES;  (* A-0-0523 -RD- Container user defined actual data B *)
                      dwUserActualDataC_i             :SM_TYPES;  (* A-0-0525 -RD- Container user defined actual data C *)
                      dwUserActualDataD_i             :SM_TYPES;  (* A-0-0527 -RD- Container user defined actual data D *)
                      dwUserActualDataE_i             :SM_TYPES;  (* A-0-0529 -RD- Container user defined actual data E *)
                      dwUserActualDataF_i             :SM_TYPES;  (* A-0-0531 -RD- Container user defined actual data F *)
END_STRUCT
END_TYPE

// IndraMotionMlc1/Application/AxisInterface/Type/Status/TE_AXIS_DIAGNOSIS
    (********** Diagnosis outputs - from motion control to logic control *****************)
    (********** Diagnose-Ausgaenge - Motion Control zur Logic Control    *****************)
// Online changes in declaration of axis-interface need too much time -> not allowed because risk of F5180006 
// InhibitOnlineChange = 0x1000000 has to be set decimal 16777216
{attribute 'signature_flag' := '16777216'} 
TYPE TE_AXIS_DIAGNOSIS EXTENDS MB_AXIS_DIAGNOSIS:

STRUCT

  (* add your extensions below here |  Erweiterungen hier einfuegen*)

  (* user extensions | Anwender Erweiterungen *)


END_STRUCT

END_TYPE

// IndraMotionMlc1/Application/AxisInterface/Type/Status/TE_AXIS_POS_STATUS
    (********* Outputs of the following axis - from motion control to logic control **********)
    (********* Achs-Ausgaenge - Motion Control zur Logic Control                    **********)
// Online changes in declaration of axis-interface need too much time -> not allowed because risk of F5180006 
// InhibitOnlineChange = 0x1000000 has to be set decimal 16777216
{attribute 'signature_flag' := '16777216'} 
TYPE TE_AXIS_POS_STATUS EXTENDS MB_AXIS_POS_STATUS:
STRUCT

	(* -> outputs of the adjusting functionality for the position
      -> Ausgaenge fuer Tippbetrieb der Position *)
    //Adjust: MB_AXIS_ADJUST_STATUS;
 
(* add your extensions below here, keep the elements above
   Erweiterungen hier einfuegen, Elemente oberhalb nicht veraendern *)

(* user extensions | Anwender Erweiterungen *)

END_STRUCT

END_TYPE

// IndraMotionMlc1/Application/AxisInterface/Type/Status/TE_AXIS_SETUP_MODE_STATUS
// Online changes in declaration of axis-interface need too much time -> not allowed because risk of F5180006 
// InhibitOnlineChange = 0x1000000 has to be set decimal 16777216
{attribute 'signature_flag' := '16777216'} 
TYPE TE_AXIS_SETUP_MODE_STATUS :
  STRUCT
    EnableAck:   BOOL; 	  (* Acknowledge setup mode  | Bestätigung Einrichtbetrieb
      - removed when _OpMode is oerwritten | - wird weggenommen, wenn _OpMode überschrieben wird *)

    HomingAck: 		BOOL; 	  (* Acknowledge Homing 
      - ModeHoming|SetAbsRef|ModesPosAbs | ModeHoming|SetAbsRef|ModesPosAbs
        finished                         | abgeschlossen                    *) 
	
  END_STRUCT
END_TYPE

// IndraMotionMlc1/Application/AxisInterface/Type/Status/TE_AXIS_STATUS_TYPE01
    (********* Outputs of the following axis - from motion control to logic control **********)
// Online changes in declaration of axis-interface need too much time -> not allowed because risk of F5180006 
// InhibitOnlineChange = 0x1000000 has to be set decimal 16777216
{attribute 'signature_flag' := '16777216'} 
TYPE TE_AXIS_STATUS_TYPE01:
  STRUCT
    (********* Outputs of the following axis - from motion control to logic control **********)

    PtrAxisData:  POINTER TO ML_AXISDATA_SM;
     (* Pointer to AxisData of this axis | Zeiger auf AxisData dieser Achse
      - Type .PtrAxisData^. for the intellisense menu | Eingabe .PtrAxisData^. fuer Auswahlmenue*)

    Admin:   TE_AXIS_ADMIN_STATUS; (* status of the axis | Achs-Status *)

    Diag:    TE_AXIS_DIAGNOSIS; (* axis diagnosis information, error, warning....
      Diagnose Informationen der Achse, Fehler, Warnung.... *)

    PosMode: TE_AXIS_POS_STATUS; (* Status operating mode positioning (absolute, rel. and add.)
      Statusmeldungen Positionierbetrieb (absolut, relativ und additiv) *)

    VelMode: TE_AXIS_VEL_STATUS; (* Status operating mode velocity control
      Statusmeldungen Geschwindigkeitsregelung (Freilauf) *)

    SyncMode: TE_AXIS_SYNC_STATUS; (* Status operating mode synchronisation (phase, vel, and cam)
      Statusmeldungen Synchronbetriebsarten (Winkelsync., Geschwindigkeitssync. und Kurvensch.)*)

    (* add your extensions below here, keep the elements above
       Erweiterungen hier einfuegen, Elemente oberhalb nicht veraendern *)
    (* user extensions | Anwender Erweiterungen *)
		(* Jog/Homing functionality | Tipp/Einrichtfunktionen *)
    SetupMode:  TE_AXIS_SETUP_MODE_STATUS;

    // AxisData for HMI (without data type "BIT")
	  AxisData_HMI:	TE_AXIS_DATA_STATUS;
	
  END_STRUCT
END_TYPE

// IndraMotionMlc1/Application/AxisInterface/Type/Status/TE_AXIS_SYNC_STATUS
    (********* Outputs of the following axis - from motion control to logic control **********)
    (********* Achs-Ausgaenge - Motion Control zur Logic Control                    **********)
// Online changes in declaration of axis-interface need too much time -> not allowed because risk of F5180006 
// InhibitOnlineChange = 0x1000000 has to be set decimal 16777216
{attribute 'signature_flag' := '16777216'} 
TYPE TE_AXIS_SYNC_STATUS EXTENDS MB_AXIS_SYNC_STATUS:
STRUCT
    // CamActiveID:      MC_CAM_ID; (* - ID of the active CamTable | - Nr. aktive Stuetzpunkt-Tab.*)

	(* - Number of the active motion profile set 0 or 1
      - Nummer des aktiven Satzes 0 oder 1 des Bewegungsprofils *)
    // ProfileActiveSet: UINT:= 0;  

	(* - Change of PhaseOffset is finished
      - Verstellung des PhaseOffset ist abgeschlossen  *)
    // PhasingSlaveDone: BOOL := FALSE; 

	(* adjusting | vertippen
      arAxisCntrl[].SyncMode.FineAdjust *)
    //AdjFineAdjust:       MB_AXIS_ADJUST_STATUS; 

	(* adjusting | vertippen
      arAxisCntrl[].SyncMode.CamShaftDistance *)
    //AdjCamShaftDistance: MB_AXIS_ADJUST_STATUS; 

	(* adjusting | vertippen
      arAxisCntrl[].SyncMode.PhaseOffset *)
    //AdjPhaseOffset:      MB_AXIS_ADJUST_STATUS;
	
  (* add your extensions below here, keep the elements above
     Erweiterungen hier einfuegen, Elemente oberhalb nicht veraendern *)

  (* user extensions | Anwender Erweiterungen *)
	AngleOffsetDone:   BOOL:= FALSE; 	// angle offset begin of profile transmission done | Winkelverschiebung Tabellenanfang Übertragung abgeschlossen  

  SyncVelocityDone:  BOOL:= FALSE;    // Synchronisation velocity transmission done | Aufsynchronisiergeschw. Übertragung abgeschlossen  

  SyncAccelerationDone: BOOL:= FALSE;	// Synchron. acceleration transmission done | Aufsynchronisierbeschleunigung Übertragung abgeschlossen
	
  PhasingMasterDone: BOOL:=FALSE;    // Change of PhaseShift is finished | Verstellung des PhaseShift ist abgeschlossen 
 
END_STRUCT

END_TYPE

// IndraMotionMlc1/Application/AxisInterface/Type/Status/TE_AXIS_VEL_STATUS
    (********* Outputs of the following axis - from motion control to logic control **********)
    (********* Achs-Ausgaenge - Motion Control zur Logic Control                    **********)
// Online changes in declaration of axis-interface need too much time -> not allowed because risk of F5180006 
// InhibitOnlineChange = 0x1000000 has to be set decimal 16777216
{attribute 'signature_flag' := '16777216'} 
TYPE TE_AXIS_VEL_STATUS  EXTENDS MB_AXIS_VEL_STATUS:
STRUCT
	(* -> outputs of the adjusting functionality for the velocity
      -> Ausgaenge fuer Tippbetrieb der Geschwindigkeit *)
    //Adjust: MB_AXIS_ADJUST_STATUS;
 
(* add your extensions below here, keep the elements above
   Erweiterungen hier einfuegen, Elemente oberhalb nicht veraendern *)

(* user extensions | Anwender Erweiterungen *)

END_STRUCT

END_TYPE

// IndraMotionMlc1/Application/OPCUA_Data_type/AxisErrorStatus_Type
TYPE AxisErrorStatus_Type :
STRUCT
	errErrorActive: BOOL;
	errFieldBus: BOOL;
	errLim2CCW: BOOL;
	errLim2CW: BOOL;
	errLimV_Err: BOOL;
	errMotComm: BOOL;
	errMotEnc: BOOL;
	errMotor: BOOL;
	errMotReady: BOOL;
	errOverride: BOOL;
	errP_DevExceed: BOOL;
	errP_RangeExceed: BOOL;
	errPosEnc: BOOL;
	errPosEnc_Fo: BOOL;
	errPower: BOOL;
	errV_DevExceed: BOOL;
	errV_MotExceed: BOOL;
END_STRUCT
END_TYPE

// IndraMotionMlc1/Application/OPCUA_Data_type/MngmtStatus_Type
TYPE MngmtStatus_Type :
STRUCT
	DscState: DscStateType;
	//ErrorStatus: MngmtErrorStatus_Type;
	FiPos: BandType;
	HHP_Az: BOOL;
	HHP_Cncted: BOOL;
	HHP_Dir_Minus: BOOL;
	HHP_Dir_Plus: BOOL;
	HHP_El: BOOL;
	HHP_Fi: BOOL;
	OnSource: BOOL;
	//PowerStatus: PowerStatus_Type;
	///TempHumidStatus: TempHumidStatus_Type;
	//WarningStatus: WarningStatus_Type;
END_STRUCT
END_TYPE

// IndraMotionMlc1/Application/OPCUA_Data_type/MotorStatus_Type
TYPE MotorStatus_Type :
STRUCT
	ErrorCode: UINT;
	mActTorq: LREAL;
	mActVelocity: LREAL;
	MotorOverload: LREAL;
	MotorTemp: LREAL;
	RateOfUtil: LREAL;
END_STRUCT
END_TYPE

// IndraMotionMlc1/Application/OPCUA_Data_type/StaticPmParam
TYPE StaticPmParam :
STRUCT
	IA:LREAL;
	CA:LREAL;
	NPAE:LREAL;
	AN:LREAL;
	AN0:LREAL;
	AW:LREAL;
	AW0:LREAL;
	ACEC:LREAL;
	ACES:LREAL;
	ABA:LREAL;
	ABphi:LREAL;
	IE:LREAL;
	ECEC: LREAL;
	ECES: LREAL;
	HECE4: LREAL;
	HESE4:LREAL;
	HECE8:LREAL;
	HESE8:LREAL;
END_STRUCT
END_TYPE

// IndraMotionMlc1/Application/OPCUA_Data_type/TableStatus_type
TYPE TableStatus_type :
STRUCT
	act_pt_act_index:UINT;(*Actual used index of the offset table*)
	act_pt_end_index:UINT;(*End index of the offset table*)
	act_pt_value_Az:LREAL;(*Actual azimuth position output for the track table (-271° to 271°)*)
	act_pt_value_El:LREAL;(*Actual elevation position output for the track table(14.8° to 90.2°)*)
	pts_Completed:BOOL;(*The tracking has reached its last table entry, the output of the function is the position of the last table entry *)
    pts_DataValid:BOOL;(*The table has valid data, a track can be started. *)
	pts_Err:BOOL;(*The tracking function reports an error *)
	pts_Interpol:InterpolType;(*Interpolation mode is 0 = Newton, 1 = Spline *)
	pts_InterpolError:BOOL;(*An error occurred during the interFIation of the table entries *)
	pts_Running:BOOL;(*The tracking has been started, the actual time has reached the start time of the table, the output position of the function is the interFIated position at the appropriate table entry *)
	pts_StartPos:BOOL;(*The output position of the function is the first table entry*)
    pts_TableAlmostFull: BOOL; (* There are less than 50 space left in the table *)
		
END_STRUCT
END_TYPE

// IndraMotionMlc1/Application/OPCUA_Data_type/TiltmeterParam
TYPE TiltmeterParam :	
STRUCT
	One:TiltmeterSubParam;
	Two:TiltmeterSubParam;
END_STRUCT
END_TYPE

// IndraMotionMlc1/Application/OPCUA_Data_type/TiltmeterSubParam
TYPE TiltmeterSubParam :	
STRUCT
    Tiltmeter_serial_no:STRING;
	tilt_temp_scale:LREAL;
	x_filt_dt:LREAL;
	x_off:LREAL;
	x_offTC:LREAL;
	x_scale:LREAL;
	x_scaleTC:LREAL;
	x_zero:LREAL;
	x_zeroTC:LREAL;
	y_filt_dt:LREAL;
	y_off:LREAL;
	y_offTC:LREAL;
	y_scale:LREAL;
	y_scaleTC:LREAL;
	y_zero:LREAL;
	y_zeroTC:LREAL;
	
	
END_STRUCT
END_TYPE

// IndraMotionMlc1/Application/OPCUA_Data_type/MngmtWarningStatus_Type
TYPE MngmtWarningStatus_Type :
STRUCT
	waAzimuth: BOOL;
	waCmd: BOOL;
	waDoorDrive: BOOL;
	waDoorEMISC: BOOL;
	waDoorPED: BOOL;
	waDoorPSC: BOOL;
	waElevation: BOOL;
	waFeedindexer: BOOL;
	waHatchAzBearing: BOOL;
	waHatchPscRoof: BOOL;
	waHornOn: BOOL;
	waMngmnt: BOOL;
	waOverTempDrive: BOOL;
	waOverTempEMISC: BOOL;
	waOverTempPED: BOOL;
	waOverTempPSC: BOOL;
	waPoint: BOOL;
	waSafe2ApproachLight: BOOL;
	waSafety: BOOL;
	waStwPin: BOOL;
	waTime: BOOL;
	waTrack: BOOL;
END_STRUCT
END_TYPE

// IndraMotionMlc1/Application/OPC_UA_Symbols_Objects/AxisSelectType
(*{attribute 'opcua.mapping.type' := ''}
{attribute 'opcua.mapping.modeluri' := 'http://skao.int/DS_ICD/'}
{attribute 'opcua.mapping.publicationdate' := '12/14/2023 00:00:00'}
{attribute 'opcua.mapping.nodeid' := 'nsu=http://skao.int/DS_ICD/;i=3007'}*)
{attribute 'linkalways'}

TYPE AxisSelectType :
(
	Unknown:=0,
    Az := 1,
	El := 2,
	Fi := 3,
	AzEl := 4
) UINT;
END_TYPE

// IndraMotionMlc1/Application/OPC_UA_Symbols_Objects/AxisStateType
(*{attribute 'opcua.mapping.type' := ''}
{attribute 'opcua.mapping.modeluri' := 'http://skao.int/DS_ICD/'}
{attribute 'opcua.mapping.publicationdate' := '12/14/2023 00:00:00'}
{attribute 'opcua.mapping.nodeid' := 'nsu=http://skao.int/DS_ICD/;i=3005'}*)
{attribute 'linkalways'}
TYPE AxisStateType :
(
	StartUp := 0,
	Standby := 1,
	Locked := 2,
	Locked_Stowed := 3,
	Activating := 4,
	Deactivating := 5,
	Standstill := 6,
	Stopping := 7,
	Slew := 8,
	Jog := 9,
	Track := 10,
	Stowed := 11
) UINT;
END_TYPE

// IndraMotionMlc1/Application/OPC_UA_Symbols_Objects/BandType
(*{attribute 'opcua.mapping.type' := ''}
{attribute 'opcua.mapping.modeluri' := 'http://skao.int/DS_ICD/'}
{attribute 'opcua.mapping.publicationdate' := '12/14/2023 00:00:00'}
{attribute 'opcua.mapping.nodeid' := 'nsu=http://skao.int/DS_ICD/;i=3020'}*)
{attribute 'linkalways'}
TYPE BandType :
(
	Optical := 0,
	Band_1 := 1,
	Band_2 := 2,
	Band_3 := 3,
	Band_4 := 4,
	Band_5a := 5,
	Band_5b := 6,
	Band_6 := 7,
	Unknown :=8
) UINT;
END_TYPE

// IndraMotionMlc1/Application/OPC_UA_Symbols_Objects/CmdResponseType
(*{attribute 'opcua.mapping.type' := ''}
{attribute 'opcua.mapping.modeluri' := 'http://skao.int/DS_ICD/'}
{attribute 'opcua.mapping.publicationdate' := '12/14/2023 00:00:00'}
{attribute 'opcua.mapping.nodeid' := 'nsu=http://skao.int/DS_ICD/;i=3003'}*)
{attribute 'linkalways'}
TYPE CmdResponseType :
(
	NoCmdAuth := 0,
	DishLocked := 1,
	CommandRejected := 2,
	CommandTimeout := 3,
	CommandFailed := 4,
	AxisNotActivated := 5,
	Stowed := 6,
	NoOfParametersError := 7,
	ParameterOutOfRange := 8,
	CommandActivated := 9,
	CommandDone := 10,
	NotImplemented :=11
) UINT;
END_TYPE

// IndraMotionMlc1/Application/OPC_UA_Symbols_Objects/DscCmdAuthorityType
(*{attribute 'opcua.mapping.type' := ''}
{attribute 'opcua.mapping.modeluri' := 'http://skao.int/DS_ICD/'}
{attribute 'opcua.mapping.publicationdate' := '12/14/2023 00:00:00'}
{attribute 'opcua.mapping.nodeid' := 'nsu=http://skao.int/DS_ICD/;i=3013'}*)
{attribute 'linkalways'}
TYPE DscCmdAuthorityType :
(
	NoAuthority := 0,
	LMC := 1,
	HHP := 2,
	EGUI := 3,
	Tester := 4
) UINT;
END_TYPE

// IndraMotionMlc1/Application/OPC_UA_Symbols_Objects/DscStateType
(*{attribute 'opcua.mapping.type' := ''}
{attribute 'opcua.mapping.modeluri' := 'http://skao.int/DS_ICD/'}
{attribute 'opcua.mapping.publicationdate' := '12/14/2023 00:00:00'}
{attribute 'opcua.mapping.nodeid' := 'nsu=http://skao.int/DS_ICD/;i=3009'} *)
{attribute 'linkalways'}
TYPE DscStateType :
(
	StartUp := 0,
	Standby := 1,
	Locked := 2,
	Stowed := 3,
	Locked_Stowed := 4,
	Activating := 5,
	Deactivating := 6,
	Standstill := 7,
	Stopping := 8,
	Slew :=9,
	Jog := 10,
	Track := 11
) UINT;
END_TYPE

// IndraMotionMlc1/Application/OPC_UA_Symbols_Objects/DscTimeSyncSourceType
(*{attribute 'opcua.mapping.type' := ''}
{attribute 'opcua.mapping.modeluri' := 'http://skao.int/DS_ICD/'}
{attribute 'opcua.mapping.publicationdate' := '12/14/2023 00:00:00'}
{attribute 'opcua.mapping.nodeid' := 'nsu=http://skao.int/DS_ICD/;i=3017'}*)
{attribute 'linkalways'}
TYPE DscTimeSyncSourceType :
(
	PTP := 0,
	NTP := 1,
	DSC := 2
) UINT:=NTP;
END_TYPE

// IndraMotionMlc1/Application/OPC_UA_Symbols_Objects/InterpolType
(*{attribute 'opcua.mapping.type' := ''}
{attribute 'opcua.mapping.modeluri' := 'http://skao.int/DS_ICD/'}
{attribute 'opcua.mapping.publicationdate' := '12/14/2023 00:00:00'}
{attribute 'opcua.mapping.nodeid' := 'nsu=http://skao.int/DS_ICD/;i=3012'}*)
{attribute 'linkalways'}
TYPE InterpolType :
(
	Spline := 0,
	Newton := 1
) UINT;
END_TYPE

// IndraMotionMlc1/Application/OPC_UA_Symbols_Objects/LoadModeType
(*{attribute 'opcua.mapping.type' := ''}
{attribute 'opcua.mapping.modeluri' := 'http://skao.int/DS_ICD/'}
{attribute 'opcua.mapping.publicationdate' := '12/14/2023 00:00:00'}
{attribute 'opcua.mapping.nodeid' := 'nsu=http://skao.int/DS_ICD/;i=3016'}*)
{attribute 'linkalways'}
TYPE LoadModeType :
(
	Append := 0,
    New := 1,
    Reset := 2
) UINT;
END_TYPE

// IndraMotionMlc1/Application/OPC_UA_Symbols_Objects/SafetyStateType
(*{attribute 'opcua.mapping.type' := ''}
{attribute 'opcua.mapping.modeluri' := 'http://skao.int/DS_ICD/'}
{attribute 'opcua.mapping.publicationdate' := '12/14/2023 00:00:00'}
{attribute 'opcua.mapping.nodeid' := 'nsu=http://skao.int/DS_ICD/;i=3006'}*)
{attribute 'linkalways'}
TYPE SafetyStateType :
(
	Running := 0,
	Stopped := 1,
	Error := 2
) UINT;
END_TYPE

// IndraMotionMlc1/Application/OPC_UA_Symbols_Objects/StowPinStatusType
(*{attribute 'opcua.mapping.type' := ''}
{attribute 'opcua.mapping.modeluri' := 'http://skao.int/DS_ICD/'}
{attribute 'opcua.mapping.publicationdate' := '12/14/2023 00:00:00'}
{attribute 'opcua.mapping.nodeid' := 'nsu=http://skao.int/DS_ICD/;i=3010'}*)
{attribute 'linkalways'}
TYPE StowPinStatusType :
(
	Unknown := 0,
    Retracted := 1,
	Retracting := 2,
	Deployed := 3,
	Deploying := 4,
	MotionTimeOut := 5
) UINT;
END_TYPE

// IndraMotionMlc1/Application/OPC_UA_Symbols_Objects/TimeSourceType
(*{attribute 'opcua.mapping.type' := ''}
{attribute 'opcua.mapping.modeluri' := 'http://skao.int/DS_ICD/'}
{attribute 'opcua.mapping.publicationdate' := '12/14/2023 00:00:00'}
{attribute 'opcua.mapping.nodeid' := 'nsu=http://skao.int/DS_ICD/;i=3011'}*)
{attribute 'linkalways'}
TYPE TimeSourceType :
(
	PTP := 0,
	NTP := 1,
	DSC := 2
) UINT;
END_TYPE

// IndraMotionMlc1/Application/OPCUA_Data_type/SafetyStatus_Type
TYPE SafetyStatus_Type :
STRUCT
	AutoStowActive: BOOL;
	Axes_InitFault: BOOL;
	EStopFi: BOOL;
	EStopHHP: BOOL;
	EStopPed: BOOL;
	EStopTurnhead: BOOL;
	HatchAzBearing: BOOL;
	HatchTurnheadRoof: BOOL;
	InterlockClearable: BOOL;  (*All interlocks have been cleared ready for Interlock_Ack command. *)
	Lim2_CCW_Az: BOOL;
	Lim2_CCW_Fi: BOOL;
	Lim2_CW_Az: BOOL;
	Lim2_CW_Fi: BOOL;
	Lim2_Dn_El: BOOL;
	Lim2_Up_El: BOOL;
	SafetyLockout_Az: BOOL;
	SafetyLockout_El: BOOL;
	SafetyLockout_Fi: BOOL;
	SafetyState: SafetyStateType;
	STO_Az: BOOL;
	STO_El: BOOL;
	STO_Fi: BOOL;
	StowPinStatus: StowPinStatusType;
END_STRUCT
END_TYPE

// IndraMotionMlc1/Application/OPCUA_Data_type/Time_cdsStatus_type
TYPE Time_cdsStatus_type :
STRUCT
	DscTimeSyncSource: DscTimeSyncSourceType;
	LeapSecPTP: UINT :=37; 
	TAIoffset: LREAL; (* TAI Offset in Seconds from SKAO Epoch*)
	TimeSourceAddrNTP: STRING := '196.10.54.57'; // This is a know NTP server accesible from the ITF
	TimeSynced: BOOL;
	UTCtoSkaEpochSec: UINT := 32;
END_STRUCT
END_TYPE

// IndraMotionMlc1/Application/OPCUA_Data_type/PointingStatus_Type
TYPE PointingStatus_Type :
STRUCT
	ActAmbTemp_East: LREAL;
	ActAmbTemp_South: LREAL;
	ActAmbTemp_West: LREAL;
	AmbTempCorrActive: BOOL;
	AmbTempCorrVal_Az: LREAL;
	AmbTempCorrVal_El: LREAL;
	BandForCorr: BandType;
	StaticPmCorrVal_Az: LREAL;
	StaticPmCorrVal_El: LREAL;
	TotalPointCorr_Az: LREAL;
	TotalPointCorr_El: LREAL;
	StaticCorrActive: BOOL;
	TiltCorrActive: BOOL;
	TiltOne_On: BOOL;
	TiltTemp_One: LREAL;
	TiltTemp_Two: LREAL;
	TiltTwo_On: BOOL;
	TiltXArcsec_One: LREAL;
	TiltXArcsec_Two: LREAL;
	TiltXFilt_One: LREAL;
	TiltXFilt_Two: LREAL;
	TiltXRaw_mV_One: LREAL;
	TiltXRaw_mV_Two: LREAL;
	TiltYArcsec_One: LREAL;
	TiltYArcsec_Two: LREAL;
	TiltYFilt_One: LREAL;
	TiltYFilt_Two: LREAL;
	TiltYRaw_mV_One: LREAL;
	TiltYRaw_mV_Two: LREAL;
	TiltCorrVal_Az: LREAL;
	TiltCorrVal_El: LREAL;
	CurrentPointing: ARRAY [0..6] OF LREAL; 
END_STRUCT
END_TYPE

// IndraMotionMlc1/Application/OPCUA_Data_type/TrackingStatus_Type
TYPE TrackingStatus_Type :
STRUCT
	act_statOffset_value_Xel:LREAL;
	act_statOffset_value_El:LREAL;
	OnSourceDev:LREAL;
	OnSourceThreshold:LREAL:=10;
    p_desired_Az:LREAL;
	p_desired_El:LREAL;
    ThresholdTimePeriod:LREAL;	
    tr_initOk:BOOL;
	tr_obj_valid:BOOL;
	tr_selPoly:BOOL;
	tr_TimeRemaining:LREAL;
	tr_valid:BOOL;
	
END_STRUCT
END_TYPE

// IndraMotionMlc1/Application/OPCUA_Data_type/PolyStatus_type
TYPE PolyStatus_type :
STRUCT
	act_PolyValue_Az: LREAL;
	act_PolyValue_El: LREAL;
	pts_Completed: BOOL;
	pts_DataValid: BOOL;
	pts_Err: BOOL;
	pts_InterpolError: BOOL;
	pts_Running: BOOL;
	pts_StartPos: BOOL;
	pts_TimeDistFault: BOOL;
	pts_TrackId_Err: BOOL;
END_STRUCT
END_TYPE

// IndraMotionMlc1/Application/OPCUA_Data_type/PowerStatus_Type
TYPE PowerStatus_Type :
STRUCT
	ActPwrCnsm: REAL; (*Power is measured at entrance to the PSC the measurement excludes the helium compressor and equipment on the Feed Indexer.*)
	cbEMISC: BOOL;
	cbFan_PSC: BOOL;
	cbHe_Comp: BOOL;
	cbPDU_Fi: BOOL;
	cbPED_Spare: BOOL;
	cbPSC_Spare: BOOL;
	CurrentPh1: REAL;
	CurrentPh2: REAL;
	CurrentPh3: REAL;
	FrequencyPh1: REAL;
	FrequencyPh2: REAL;
	FrequencyPh3: REAL;
	LowPowerActive: BOOL:= FALSE; (*Low power mode active: True=Low power, False=Normal.*)
	PowerFactor: REAL;
	VoltagePh1: REAL;
	VoltagePh2: REAL;
	VoltagePh3: REAL;
	SpdFnctnl_PDU1:BOOL;
	SpdFnctnl_PDU2:BOOL;
END_STRUCT
END_TYPE

// IndraMotionMlc1/Application/OPCUA_Data_type/AxisWarning_Type
TYPE AxisWarning_Type :
STRUCT
	waParamFault:BOOL;
	waOverride :BOOL;
	waMotReady :BOOL;
	waMotWarn :BOOL;
	waMmaxExceeded :BOOL;
	waLim1CW:BOOL;
	waLim1CCW:BOOL;
	waLimSoftCW:BOOL;
	waLimSoftCCW:BOOL;
	waPosEncWarn:BOOL;
	waStowPinsDep:BOOL;
	waVelLimit :BOOL;
END_STRUCT
END_TYPE

// IndraMotionMlc1/Application/OPCUA_Data_type/MngmtErrorStatus_Type
TYPE MngmtErrorStatus_Type :
STRUCT
	errAuthLost: BOOL; (*The actual control authority is not communicating. The dish structure will go to STANDBY If no connection is made within the AutoStow timeout the Dish will stow automatically.*)
	errAzimuth: BOOL; 
	errCmd: BOOL;
	errElevation: BOOL;
	errFeedindexer: BOOL;
	errGeneral: BOOL;
	errMngmnt: BOOL;
	errPoint: BOOL;
	errPwr24VDC: BOOL;
	errPwr400VAC: BOOL;
	errPwr600VDC: BOOL;
	errPwrMeterComms: BOOL;
	errSafety: BOOL;
	errStwPin: BOOL;
	errTiltOneComms: BOOL;
	errTiltOneIoUnit: BOOL;
	errTiltTwoComms: BOOL;
	errTiltTwoIoUnit: BOOL;
	errTime: BOOL;
	errTrack: BOOL;
END_STRUCT
END_TYPE

// IndraMotionMlc1/Application/OPCUA_Data_type/TempHumidStatus_Type
TYPE TempHumidStatus_Type :
STRUCT
	HumidDriveCab: REAL;
	HumidPSC_Inlet: REAL;
	HumidPSC_Outlet: REAL;
	TempDriveCab: REAL;
	TempEMISC_Outlet: REAL;
	TempPSC_Inlet: REAL;
	TempPSC_Outlet: REAL;
END_STRUCT
END_TYPE

// IndraMotionMlc1/Application/OPCUA_Data_type/NamePlate_Type
TYPE NamePlate_Type :
STRUCT
	DishId:STRING:= 'ITF_DEV';
	DishStructureSerialNo:STRING:='ITF 1';
    DscSoftwareVersion:STRING:= '0.0.3';
	IcdVersion: STRING := '301-000000-082 Rev 2A';
	RunHours:LREAL;
	TotalDist_Az:LREAL;
	TotalDist_El_deg:LREAL;
	TotalDist_El_m:LREAL;
	TotalDist_Fi:LREAL;
	
END_STRUCT
END_TYPE

// IndraMotionMlc1/Application/OPCUA_Data_type/CommandArbiter_Status_Type
TYPE CommandArbiter_Status_Type :
STRUCT
	DscCmdAuthority: DscCmdAuthorityType; (* the authority for DSC control now 0 NoAuthority 1 LMC 2 HHP 3 EGUI*)
	LastCmdResponse: CmdResponseType;    (* Command response of the last command *)
	LastLoadMode: LoadModeType; 		// Last loadmode Called
	LastTiltOn:   TiltOnType;       	 // Last Tiltmeter switched on 
	AxisSelect: AxisSelectType;     	// Last Selected Axis
	
	
END_STRUCT
END_TYPE

// IndraMotionMlc1/Application/OPCUA_Data_type/AxisGeneralStatus_Type
TYPE AxisGeneralStatus_Type :
STRUCT
	Active: BOOL;
	AllActive: BOOL;
	AxisMoving: BOOL;
	AxisState: AxisStateType;
	encBoxOp: BOOL;
	EStop: BOOL;
	Exceed: BOOL;
	InitOk: BOOL;
	LimOverride: BOOL;
	p_Act: LREAL;
	p_Dev: LREAL;
	p_Enc: LREAL;
	p_PointCorr: LREAL;
	p_Set: LREAL;
	p_Shape: LREAL;
	posDevOk: BOOL;
	Ready: BOOL;
	Reset: BOOL;
	SectorSw: BOOL;
	StowPos_Minus: LREAL:= -0.007;
	StowPos_Plus: LREAL:= 0.007;
	TorqueBias:LREAL;
	TorqueTotal:LREAL;
	v_Act: LREAL;
	v_SetMax: LREAL;
	v_Shape: LREAL;
	
	
END_STRUCT
END_TYPE

// IndraMotionMlc1/Application/OPC_UA_Symbols_Objects/TiltOnType
{attribute 'qualified_only'}

TYPE TiltOnType :
(
	Off :=0,
	TiltmeterOne :=1,
	TiltmeterTwo :=2
)UINT;
END_TYPE

// IndraMotionMlc1/Application/MlcVarGlobal
(* Automatically generated code by XLC/MLC. *)
(* Please don't edit, the code will be overwritten. For usercode use UserVarGlobal! *)
{attribute 'linkalways'}
{attribute 'analysis' := '-33'}
VAR_GLOBAL CONSTANT

(*Virtual axis "drive1" with axis number 1*)
drive1: AXIS_REF :=(CntrlNo:=LOCAL_CNTRL,AxisNo:=AXIS_1);

(*Virtual axis "drive2" with axis number 2*)
drive2: AXIS_REF :=(CntrlNo:=LOCAL_CNTRL,AxisNo:=AXIS_2);

(*Virtual axis "drive3" with axis number 3*)
drive3: AXIS_REF :=(CntrlNo:=LOCAL_CNTRL,AxisNo:=AXIS_3);

(*Virtual axis "Drive4" with axis number 4*)
Drive4: AXIS_REF :=(CntrlNo:=LOCAL_CNTRL,AxisNo:=AXIS_4);

(*Virtual axis "Drive5" with axis number 5*)
Drive5: AXIS_REF :=(CntrlNo:=LOCAL_CNTRL,AxisNo:=AXIS_5);

(*Virtual axis "Drive6" with axis number 6*)
Drive6: AXIS_REF :=(CntrlNo:=LOCAL_CNTRL,AxisNo:=AXIS_6);

(*Virtual axis "v_azimuth" with axis number 7*)
v_azimuth: AXIS_REF :=(CntrlNo:=LOCAL_CNTRL,AxisNo:=AXIS_7);

(*Virtual axis "v_elevation" with axis number 8*)
v_elevation: AXIS_REF :=(CntrlNo:=LOCAL_CNTRL,AxisNo:=AXIS_8);

(*Virtual axis "v_FeedIndexer" with axis number 9*)
v_FeedIndexer: AXIS_REF :=(CntrlNo:=LOCAL_CNTRL,AxisNo:=AXIS_9);

(*Virtual axis "v_time_master" with axis number 10*)
v_time_master: AXIS_REF :=(CntrlNo:=LOCAL_CNTRL,AxisNo:=AXIS_10);


END_VAR

// IndraMotionMlc1/Application/Global_Variables
VAR_GLOBAL
(*<<<<<<<<<<<<<<<<<<< Cold start variables >>>>>>>>>>>>>>>>>>>>>>>>>>>>>>>>>>>>>>>*)
   b_startup:BOOL:=1;
	

(*<<<<<<<<<<<<<<<<<<<<<<<<<<<<<< Stopping Commands and variables>>>>>>>>>>>>>>>>>>>>>>>>>>>>>>>>>*)
    b_stop_Az:BOOL; (*The command of stop the motion of Azimuth*)
	b_stop_El:BOOL; (*The command of stop the motion of Elevation*)
	b_stop_Fi:BOOL; (*The command of stop the motion of Feed Indexer*)
	b_stop_act_Az: BOOL; // Az busy stopping
	b_stop_act_El: BOOL; // El busy stopping
	b_stop_act_Fi: BOOL; // Fi busy stopping
	
(*<<<<<<<<<<<<<<<<<<<<<<<<<<<<<< Activating and Deactivating>>>>>>>>>>>>>>>>>>>>>>>>>>>>>>>>>*)
   b_activate_Az:BOOL:=0;
   b_activate_El:BOOL:=0;
   b_activate_Fi:BOOL:=0;
   b_deactivate_Az:BOOL:=0;
   b_deactivate_El:BOOL:=0;
   b_deactivate_Fi:BOOL:=0;
   b_Move2Band_deactivate:BOOL:=0;   
 
	
(*<<<<<<<<<<<<<<<<<<<<<<<<<<<<<<<<<<<<<< Stow >>>>>>>>>>>>>>>>>>>>>>>>>>>>>>>>>>>>>>>>>>>>>>>>>*)
    b_stow:BOOL;(*the command of stowing the antenna at 90_degrees*)
	b_stow_pulse:BOOL; // pulse to start stowing from stow method
	b_unlock: BOOL;(*the command of unlock the antenna*)
	b_stow_lock_allow :BOOL; // The azimuth is in a position where the stow pin can be inserted.
	b_lock_off: BOOL;(*power off after arriving at the stow position *)
	b_lock_off_m: BOOL;(*power off after arriving at the maintain position *)
	b_maintain_lock:BOOL;(*the signal means that antenna is locked at maintain position*)
	b_stow_lock:BOOL;(*the signal means that antenna is locked at stow position*)
	b_move_0_done: BOOL;(* the azimuth had move to the stow position*)
	b_move_90_done: BOOL;(* the elevation had move to the stow position*)
	b_move_20_done: BOOL;(* the elevation had move to the Maintenance position*)
	b_manual_stow: BOOL; // for move stowpin method to enter stowpin deploy ladder logic.
	b_UPS_Stow: BOOL:=0; // Stow under UPS drive

(*<<<<<<<<<<<<<<<<<<<<<<<<<<<<<<<<<<<< Clear Err >>>>>>>>>>>>>>>>>>>>>>>>>>>>>>>>>>>>>>>>>>*)	
    //b_pwr_on:BOOL;
	//b_pwr_off: BOOL;
	b_clear_err: BOOL;
	b_clear_err_Az: BOOL;
	b_clear_err_El: BOOL;
	b_clear_err_Fi: BOOL;
	
(*<<<<<<<<<<<<<<<<<<<<<<<<<<<<Safety and interlock related >>>>>>>>>>>>>>>>>>>>>>>>>>>>>>*)
    
	b_in_Estop:BOOL;     (* one of the Estop still active*)
	b_Estop_active:BOOL; (* signbit of Estop active, need InterlockAck to reset*)
	b_in_interlock:BOOL; (* one of the Interlock still active*)
	b_in_interlock_Az:BOOL; 
	b_in_interlock_El:BOOL;
	b_in_interlock_Fi:BOOL;
	b_Interlock_active:BOOL;(* signbit of Interlock active, need InterlockAck to reset*)	

    b_interlock_active_Az: BOOL;
	b_interlock_active_El: BOOL;
	b_interlock_active_Fi: BOOL;
	

	
(*<<<<<<<<<<<<<<<<<<<<<<<<<<<<<<<< Tracking >>>>>>>>>>>>>>>>>>>>>>>>>>>>>>>>>>>>>>>>>>>>>>*)
   b_track_start:BOOL;  // From TrackStart method used to start track along with l_start_time
   lr_track_start_time: LREAL; // Time when the track should start. 
   t_onsource_dev_filt: TIME:= t#10s; // Time constant for onsource deviation filter. 
   
   
   
   
(*<<<<<<<<<<<<<<<<<<<<<<<<<<<<<< Motion >>>>>>>>>>>>>>>>>>>>>>>>>>>>>>>>>>>>>>>>>>>>>>>*)
   b_track_on: BOOL;(*the command of running trajectory*)
   b_slew_az_el: BOOL:= FALSE;
   b_goto_rel: BOOL;
   r_vel_max_Az: REAL := gc_r_vel_max_Az;
   r_vel_max_El: REAL := gc_r_vel_max_El;
   r_vel_max_Fi: REAL := gc_r_vel_max_Fi;
   r_goto_acc_Az: REAL := gc_r_goto_acc_Az;
   r_goto_acc_El: REAL := gc_r_goto_acc_El; 
   r_goto_acc_Fi: REAL := gc_r_goto_acc_Fi;
		
  

(*<<<<<<<<<<<<<<<<<<<<<<<<<<<<<<TCP commands and variables>>>>>>>>>>>>>>>>>>>>>>>>>>>>>>>>>*)
	
	b_track_on_first:BOOL;(*judge the first point can be reached*)
	b_on_track_mode:BOOL;(*switch to the control mode of track*)
	b_Track_Pause:BOOL;(*the command of track pause*)
	b_SCC_Stop:BOOL;(*the command of stop the motion*)
	b_SCC_goto: BOOL;(*the command of goto a fixed position for all axises*)
	b_scc_goto_az: BOOL;(*the command of goto a fixed position for AZ*)
	b_scc_goto_el: BOOL;(*the command of goto a fixed position for EL*)
	b_scc_goto_FI: BOOL;(*the command of goto a fixed position for FI*)
	b_scc_vel:BOOL;(*the command of run in a fixed velocity for all axises*)
	b_SCC_STOW:BOOL;(*the command of stowing the antenna at 90_degrees*)
	b_SCC_UNLOCK: BOOL;(*the command of unlock the antenna*)
	b_SCC_maintain: BOOL;(*the command of stowing the antenna at 20_degrees*)
	b_scc_enable_on:BOOL;(*the command to enable all the drives*)
	b_scc_enable_off:BOOL;(*the command to disable all the drives*)
	b_scc_enable_start: BOOL;(*the command for start to enable all the drives*)
	b_on_write:BOOL:=TRUE;(*wrige cycle when it on*)
	b_off_write:BOOL:=FALSE;(*wrige cycle when it off*)
	ui_Length_Reply:UINT;(*the length of the reply message*)
	STR_GSTAT_M: STRING(1500);(*the middle variable of reply for Gstat command*)
	STR_K2STAT_M: STRING(255);(*the middle variable of reply for K2stat command for E-stop*)
	STR_K4STAT_M: STRING(255);(*the middle variable of reply for K4stat command for diagnostication*)
	STR_K5STAT_M: STRING(255);(*the middle variable of reply for K5stat command for limit check*)
	master_status:DWORD;
	r_offset_az: LREAL;
	r_offset_el: LREAL;
	r_offset_el_program: LREAL;
	b_offset: BOOL;
	lockstand:BOOL;
	b_M_time_done: BOOL;(*NTP source time synced*)
	b_no_SetDateTime: BOOL:=TRUE; // Prevents systime update if DSC is selected as time source
	
(*<<<<<<<<<<<<<<<<<<<<<<<<<<<<<<<<<<<NTP>>>>>>>>>>>>>>>>>>>>>>>>>>>>>>>>>>>>>>>>>>>>>>>>>>*)
	b_ntp_update_start:BOOL;(*the command of NTP update *)
	B_NTP_NEED_UPDATE:BOOL;(*the system time needs update,and the system time is checked every hour*)
	lr_MJD_current: LREAL;(*the current MJD time variable*)
	lr_TAIoffset_Current:LREAL (*the current TAI offset variable*);
	di_MJD_day:DINT;(*the current day of MJD*)

	i_num_quarter: DINT;(*the cycle number of V_time_master axis*)
	
(*<<<<<<<<<<<<<<<<<<<<<<<<<<<<<<<stack manager>>>>>>>>>>>>>>>>>>>>>>>>>>>>>>>>>>>>>>>>>>>>*)
	r_track_error:ARRAY [1..3] OF LREAL;(*track following error*)
	//i_num_stack_left: UINT;(*trajectory points number*)
	i_num_stack_left: INT;(*trajectory points number*)
	track_table: ARRAY [1..gc_stack_length] OF Stack_buffer;(*the time and positions of the point on the trajectory*)
	i_Start:INT:=1;(*the first number of trajectory*)
	i_End: INT:=1;(*the last number of trajectory*)
	i_total:INT:=gc_stack_length;(*the capability of the sack*)
	b_track_overspeed_az: BOOL:=0;(*the signbit of az track overspeed*)
	b_track_overspeed_el: BOOL:=0;(*the signbit of az track overspeed*)
	b_track_overspeed_FI: BOOL:=0;(*the signbit of az track overspeed*)
	
(*<<<<<<<<<<<<<<<<<<<<<<<<<<<<Inport variables on MLC>>>>>>>>>>>>>>>>>>>>>>>>>>>>>>>>>>>>>*)
(*----------------------------------------------------------------------------------------*)
(*         Modified for testing comment out this section for production                   *)
(*----------------------------------------------------------------------------------------*)

	b_HMV_warning : BOOL;(*the warning of HMV*)     
	b_HMV_UD : BOOL;(*the UD of HMV*)              
	b_stow_pin_limit_lock : BOOL:=1;(*locked*) // Stow pin deployed limit active
	b_stow_pin_limit_unlock : BOOL:=0;(*unlocked*) // Stow pin retracted limit active
	b_DriveCabinetDoor_Estop :BOOL:=0;(*the estop of DriveCabinetDoor*)
	b_DSDoor_Estop  :BOOL:=0;(*the estop of DSDoor*)
	b_PSCDoor_Estop :BOOL:=0;(*the estop of DPSCDoor*)
	b_AZ_Hatch  :BOOL:=0;(*the estop of AZ_Hatch*)
	b_Turnhead_Hatch  :BOOL:=0;(*the estop of Turnhead_Hatch*)
	b_DS_Estop  :BOOL:=0;(*the estop of DS*)
	b_Turnhead_Estop  :BOOL:=0;(*the estop of Turnhead*)
	b_FI_Estop  :BOOL:=0;(*the estop of FI*)

	b_HHP_Connected : BOOL:=0;      
	b_HHP_AZ : BOOL:=0;
	b_HHP_EL : BOOL:=0;
	b_HHP_Interlock : BOOL:=0;
	b_HHP_move_cw_slow : BOOL:=0;
	b_HHP_move_ccw_slow : BOOL:=0;
	b_HHP_move_cw_fast : BOOL:=0;
	b_HHP_move_ccw_fast : BOOL:=0;
	
	b_HHP_ENABLE  :BOOL:=0;
	b_HHP_STOW  :BOOL:=0;
	b_HHP_Motor_UNLOCK  :BOOL:=0;
	b_HHP_Disable  :BOOL:=0;
	b_EMISCDoor_Estop  :BOOL:=0; (*the estop of EMISCDoor*)
	b_HHP_Estop :BOOL:=0;(*the estop of HHP*)
	b_MAIN_PD_Compressor_breaker_on  :BOOL:=1;
	b_MAIN_PD_MAIN_lighting_on  :BOOL:=1;
	
	b_MAIN_PD_FI_Breaker_on :BOOL:=1;
	b_MAIN_PD_spare :BOOL:=1;
	b_PSC_PD_Light_Breaker_on :BOOL:=1;
	b_PSC_PD_EMISC_Breaker_on :BOOL:=1;
	b_PSC_PD_FAN_Breaker_on  :BOOL:=1;
	b_PSC_PD_spare :BOOL:=1;
	b_FI_PD_FI1_Breaker_on :BOOL:=1;
	b_FI_PD_FI2_Breaker_on  :BOOL:=1;
	
	b_Lock_Out_Az: BOOL:=0;
	b_Lock_Out_El: BOOL:=0;
	b_Lock_Out_Fi: BOOL:=0;
	
(*
(*<<<<<<<<<<<<<<<<<<<<<<<<<<<<Inport variables on MLC>>>>>>>>>>>>>>>>>>>>>>>>>>>>>>>>>>>>>*)
	b_HMV_warning AT %IX0.4 : BOOL;(*the warning of HMV*)     
	b_HMV_UD AT %IX0.5 : BOOL;(*the UD of HMV*)              
	b_stow_pin_limit_lock AT %IX0.6 : BOOL;(*locked*) // Stow pin deployed limit active
	b_stow_pin_limit_unlock AT %IX0.7 : BOOL;(*unlocked*) // Stow pin retracted limit active
	b_DriveCabinetDoor_Estop AT %IX1.0 :BOOL;(*the estop of DriveCabinetDoor*)
	b_DSDoor_Estop AT %IX1.1 :BOOL;(*the estop of DSDoor*)
	b_PSCDoor_Estop AT %IX1.2 :BOOL;(*the estop of DPSCDoor*)
	b_AZ_Hatch AT %IX1.3 :BOOL;(*the estop of AZ_Hatch*)
	b_Turnhead_Hatch AT %IX1.4 :BOOL;(*the estop of Turnhead_Hatch*)
	b_DS_Estop AT %IX1.5 :BOOL;(*the estop of DS*)
	b_Turnhead_Estop AT %IX1.6 :BOOL;(*the estop of Turnhead*)
	b_FI_Estop AT %IX1.7 :BOOL;(*the estop of FI*)

	b_HHP_Connected AT %IX2.0: BOOL;      
	b_HHP_AZ AT %IX2.2: BOOL;
	//b_HHP_EL AT %IX2.4: BOOL;
	b_HHP_EL : BOOL;
	b_HHP_FI AT %IX2.4: BOOL;	

	b_HHP_Interlock AT %IX2.6: BOOL;
	b_HHP_move_cw_slow AT %IX2.1: BOOL;
	b_HHP_move_ccw_slow AT %IX2.3: BOOL;
	b_HHP_move_cw_fast AT %IX2.5: BOOL;
	b_HHP_move_ccw_fast AT %IX2.7: BOOL;
	
	b_HHP_ENABLE AT %IX3.0 :BOOL;
	b_HHP_STOW AT %IX3.2 :BOOL;
	b_HHP_Motor_UNLOCK AT %IX3.4 :BOOL;
	b_HHP_Disable AT %IX3.6 :BOOL;
	b_EMISCDoor_Estop AT %IX3.1 :BOOL; (*the estop of EMISCDoor*)
	b_HHP_Estop AT %IX3.3 :BOOL;(*the estop of HHP*)
	b_MIAN_PD_Compressor_breaker_on AT %IX3.5 :BOOL;
	b_MIAN_PD_MAIN_lighting_on AT %IX3.7 :BOOL;
	
	b_MIAN_PD_FI_Breaker_on AT %IX4.0 :BOOL;
	b_MIAN_PD_spare AT %IX4.2 :BOOL;
	b_PSC_PD_Light_Breaker_on AT %IX4.4 :BOOL;
	b_PSC_PD_EMISC_Breaker_on AT %IX4.6 :BOOL;
	b_PSC_PD_FAN_Breaker_on AT %IX4.1 :BOOL;
	b_PSC_PD_spare AT %IX4.3 :BOOL;
	b_FI_PD_FI1_Breaker_on AT %IX4.5 :BOOL;
	b_FI_PD_FI2_Breaker_on AT %IX4.7 :BOOL;
	
	b_Lock_Out_Az AT %IX0.0: BOOL;
	b_Lock_Out_El AT %IX0.1: BOOL;
	b_Lock_Out_Fi AT %IX0.2: BOOL;
	
	b_PED_Door At %IX??: Bool;
	
	
*)

(*<<<<<<<<<<<<<<<<<<<<<<<<<<<<<<<<<<Outport variables On MLC>>>>>>>>>>>>>>>>>>>>>>>>>>>>>>>>*)
	b_power_on AT %QX0.0:BOOL;(*power the drives*)
	b_stow_pin_deploy AT %QX0.1:BOOL;(* activates stow pin deploy*)
	b_stow_pin_retract AT %QX0.2:BOOL;(*activates stow pin retract*)
	b_output_spare AT %QX0.3:BOOL;(*spare*)
	b_Alarm AT %QX0.4:BOOL;(*alarm on*)
	b_Horn AT %QX0.5:BOOL;(*horn on*)
	
	MAIN_PD_Compressor_Control_on AT %QX1.0:BOOL;
	PSC_PD_FAN_Control_on AT %QX1.1:BOOL;
	MAIN_PD_Indexer_Control_on AT %QX1.2:BOOL;
	PSC_PD_FAN_Spare_on AT %QX1.3:BOOL;
	MAIN_PD_Spare_Control_on AT %QX1.4:BOOL;
	PSC_PD_EMISC_Control_on AT %QX1.6:BOOL;
(*<<<<<<<<<<<<<<<<<<<<<<<<<<<<<<<<<I/O on Drives>>>>>>>>>>>>>>>>>>>>>>>>>>>>>>>>>>>>>>>>>>>>>*)
	b_estop_dr:BOOL;(*the action of pedestal estop*)
	b_estop_az :BOOL;(*the action of azimuth cable estop*)
	b_estop_el: BOOL;(*the action of elevation box estop*)
	b_estop_FI:BOOL;(*the action of FeedIndexer cable estop*)  
(*<<<<<<<<<<<<<<<<<<<<<<<<<<<<<<<the position of all the axises>>>>>>>>>>>>>>>>>>>>>>>>>>>*)
	r_pos_az:LREAL;(*real position of azimuth*)
	r_pos_el:LREAL;(*real position of elevation*)
	r_pos_FI:LREAL;(*real position of FeedIndexer*)
	r_pos_az_v:LREAL;(*the position of vitual azimuth axis*)
	r_pos_el_v:LREAL;(*the position of vitual elevation axis*)
	r_pos_FI_v:LREAL;(*the position of vitual FeedIndexer axis*)
(*<<<<<<<<<<<<<<<<<<<move azimuth by the switch on pannel>>>>>>>>>>>>>>>>>>>>>>>>>>>>>>>>>>>>*)
	b_clockwise_Az :BOOL;
    b_cclockwise_Az :BOOL;
	b_speed_Az :BOOL;
	b_enable_Az: BOOL;
	//b_activate_Az:BOOL;
(*<<<<<<<<<<<<<<<<<<<<<move elevation by the switch on pannel>>>>>>>>>>>>>>>>>>>>>>>>>>>>>>>>*)
	b_up_el :BOOL;
    b_down_el :BOOL;
	b_speed_el :BOOL;
	b_enable_el: BOOL;
	//b_activate_el:BOOL;
(*<<<<<<<<<<<<<<<<<<<<<<move FeedIndexer by the switch on pannel>>>>>>>>>>>>>>>>>>>>>>>>>>>>*)
	b_clockwise_FI :BOOL;
    b_cclockwise_FI :BOOL;
	b_speed_FI :BOOL;
	b_enable_FI: BOOL;
	//b_activate_FI:BOOL;
	
(*FP_S_0_0084,Torque force feedback value*)
	r_torque_1: REAL;
	r_torque_2: REAL;
	r_torque_3: REAL;
	r_torque_4: REAL;
	r_torque_5: REAL;
	r_torque_6: REAL;
(*<<<<<<<<<<<<<<<<<<<<<<<<<<<<<<<the limit variables>>>>>>>>>>>>>>>>>>>>>>>>>>>>>>>>>>>>>>>>>*)
	b_limit_cw_az:BOOL;(*the first hardware clockwise limit of azimuth*)
	b_limit_ccw_az:BOOL;(*the first hardware counter-clockwise limit of azimuth*)
	b_limit_final_cw_az: BOOL;(*the second hardware limit of azimuth cw*)
	b_limit_final_ccw_az: BOOL;(*the second hardware limit of azimuth ccw*)
	b_limit_cw_el:BOOL;(*the first hardware upper limit of elevation up*)
	b_limit_ccw_el:BOOL;(*the first hardware underside limit of elevation down*)
	b_limit_final_cw_el: BOOL;(*the second hardware limit of elevation up *)
	b_limit_final_ccw_el: BOOL;(*the second hardware limit of elevation down*)
	
	b_limit_cw_FI:BOOL;(*the first hardware clockwise limit of FeedIndexer*)
	b_limit_ccw_FI:BOOL;(*the first hardware counter-clockwise limit of FeedIndexer*)
	b_limit_final_cw_FI: BOOL;(*the second hardware limit of FeedIndexer cw*)
	b_limit_final_ccw_FI: BOOL;(*the second hardware limit of FeedIndexer ccw*)
(*<<<<<<<<<<<<<<<<<<<<<<<<<<<<<<<<<<<<<Power and Enable>>>>>>>>>>>>>>>>>>>>>>>>>>>>>>>>>>>>>>*)
	b_enable_az_1: BOOL;(*the enable of drive 1*)
	b_enable_az_2: BOOL;(*the enable of drive 2*)
	b_enable_el_3: BOOL;(*the enable of drive 3*)
	b_enable_el_4: BOOL;(*the enable of drive 4*)
	b_enable_FI_5: BOOL;(*the enable of drive 5*)
	b_enable_FI_6: BOOL;(*the enable of drive 6*)
	b_remote_on_run: BOOL;(*It means all the drive are ok for running*)
(*<<<<<<<<<<<<<<<<<<<<<<<<<<<<<<<<<<<<<<<<PID>>>>>>>>>>>>>>>>>>>>>>>>>>>>>>>>>>>>>>>>>>>>>>>>*)
	b_PID_in_az: BOOL;(* the antibacklash is ok,so that azimuth can be moved*)
	b_PID_in_el: BOOL;(* the antibacklash is ok,so that elevation can be moved*)
	b_PID_in_FI: BOOL;(* the antibacklash is ok,so that FIarazation can be moved*)
	b_gearin_2_done: BOOL;(*drive 1 and 2 are synchronous with v_azimuth*)
	b_gearin_4_done: BOOL;(*drive 3 and 4 are synchronous with v_elevation*)
	b_gearin_6_done: BOOL;(*drive 5 and 6 are synchronous with v_FeedIndexer*)
	b_gearinpos_5_done: BOOL;(*drive 5 is synchronous with v_FeedIndexer,so that FeedIndexer can be moved*)

(*<<<<<<<<<<<<<<<<<<<<<<<<<<<<<<<<<<<<<<<black box>>>>>>>>>>>>>>>>>>>>>>>>>>>>>>>>>>>>>>>>>>>*)
	b_send_blackbox_admin: BOOL;(*if true,the TCP sending for blackbox is allowed*)
	i_speed_1: REAL;(*the velocity feedback value of motor1*)
	i_speed_2: REAL;(*the velocity feedback value of motor1*)
	i_speed_3: REAL;(*the velocity feedback value of motor3*)
	i_speed_4: REAL;(*the velocity feedback value of motor1*)
	i_speed_5: REAL;(*the velocity feedback value of motor5*)
	i_speed_6: REAL;(*the velocity feedback value of motor1*)
	i_pos_cmd_1: REAL;
(**********************************get the MLC address*************************************)
	str_MLC_ip: STRING :='127.0.0.1';(*IP number in MLC*)
	fb_read_MLC_ip: MB_ReadStringParameter;
	str_1xx: STRING;(*the last 3 number of IP*)
(*********************************Zero Velocity****************************************)
	b_goto_Az_done: BOOL;
	b_goto_El_done: BOOL;
	b_goto_FI_done: BOOL;
(***********************************Trajectory ************************************)

	b_write_az: BOOL;
	b_write_el: BOOL;
	b_write_FI: BOOL;
	r_limit_s91: REAL;
	b_write_az_done: BOOL;
	b_write_el_done: BOOL;
	b_write_FI_done: BOOL;
	b_open_channel_az: BOOL;
	b_open_channel_el: BOOL;
	b_open_channel_FI: BOOL;
	b_open_channel_az_done: BOOL;
	b_open_channel_el_done: BOOL;
	b_open_channel_FI_done: BOOL;
	
(************************************useless****************************************)	
	//b_stow :BOOL;(*to lock antenna at 90degrees*)
	b_maintain :BOOL;(*to lock antenna at 20degrees*)
	b_remote_on:BOOL;(*in the remote mode*)
	b_local_on  :BOOL;(*in the local mode*)
	b_estop_mc:BOOL;(*the action of pannel estop*)
	b_zone_az: BOOL:= TRUE;(*the zone signal of azimuth*)
	b_power_Az :BOOL;(*close the azimuth contactor*)
	b_power_el :BOOL;(*close the elevation contactor*)
	b_power_FI :BOOL;(*close the FeedIndexer contactor*)
	b_led_unlock: BOOL;(*light the LED on pannel for unlock*)
	b_led_lock : BOOL;(*light the LED on pannel for lock*)

	
(*FP_P_0_0440,Actual output current value absolute value*)
	r_current_1: LREAL;
	r_current_2: LREAL;
	r_current_3: LREAL;
	r_current_4: LREAL;
	r_current_5: LREAL;
	r_current_6: LREAL;
(*FP_S_0_0383,Motor temperature*)
	r_temp_motor1: LREAL;
	r_temp_motor2: LREAL;
	r_temp_motor3: LREAL;
	r_temp_motor4: LREAL;
	r_temp_motor5: LREAL;
	r_temp_motor6: LREAL;	

    b_encoder_ok_az:BOOL;
	b_encoder_ok_FI:BOOL;
	B_system_encoder_OK:BOOL;
	B_encoder_home_d1:BOOL;
	B_encoder_home_d5:BOOL;
	b_home_d1: BOOL;
	b_home_d5: BOOL;
	status_code1:STRING;
	status_code2:STRING;
	status_code3:STRING;
	status_code4:STRING;
	status_code5:STRING;
	status_code6:STRING;
	b_permit_new_file:BOOL;
	r_test1:LREAL;
	r_test2:LREAL;
	r_test3:LREAL;
	b_move_to_start1: BOOL;
	b_move_to_start5: BOOL;
	i_receive_cmd:UINT:=0;
	i_excute_cmd:UINT:=0;
	last_command:STRING:='00';
(*FP_s_0_0189,following error*)
	r_following_11: LREAL;
	r_following_33: LREAL;
	r_following_1: LREAL; // Azimuth
	r_following_3: LREAL; // Elevation
	r_following_5: LREAL;
	r_following_radius_asec: REAL; // Following radius in arcseconds
		
	RATIO_OUTPUT: UINT := 1;
	RATIO_INPUT: UINT := 1;
	b_gearin_3_done:BOOL;
	gear_ratio:LREAL;
	r_pos_az_1: LREAL;
	r_pos_el_1: LREAL;
	r_pos_az_modify: LREAL;
	r_pos_el_modify: LREAL;
	
	rPosdiff: LREAL;
	roldposition:LREAL;
	r_length: LREAL;
	
	DeltaB: LREAL;
	r_length_count:LREAL;
	Inir_Length: LREAL;
	r_length_Distance: LREAL;
	r_length_Distance_1: LREAL;
	r_pos_motor3: LREAL;
	b_scc_vel1_temp: BOOL;
	
	r_goto_Az: REAL;// Relative position change 
	r_goto_v_Az: REAL; (* Velocity input of goto*)
	b_moving_Az: BOOL; // Azimuth is moving
	b_start_goto_Az:BOOL:= FALSE;
	b_start_goto_az_tcp : BOOL; // Separates goto for tcp to prevent confusion with OPCUA
		
	r_goto_El: REAL; // Relative position change 
	r_goto_v_El: REAL; (* Velocity input of goto*)
	b_moving_El: BOOL; // Elevation is moving
	b_start_goto_El:BOOL; 
	
	r_goto_Fi: REAL; // Relative position change 
	r_goto_v_Fi: REAL; (* Velocity input of goto*)
	b_moving_Fi: BOOL; // Feed Indexer is moving
	b_start_goto_Fi:BOOL; 
	
	r_goto_El_abs: LREAL;
	r_command_vel:LREAL;
	b_in_positionMode: BOOL;
	r_goto_Az_I: REAL;(*input value of goto*)
	
	r_goto_El_I: LREAL;
	r_goto_Fi_I: REAL;
		
	b_first_pos_done:BOOL;
	b_second_pos_done:BOOL;
	b_3rd_pos_done:BOOL;
	b_4th_pos_done:BOOL;
	b_5th_pos_done:BOOL;
	b_6th_pos_done:BOOL;
	b_7th_pos_done:BOOL;
	b_8th_pos_done:BOOL;
	b_9th_pos_done:BOOL;
	b_10th_pos_done:BOOL;
	i_adjust_count:INT:=0;
	adjust_delay:BOOL;
	i_closeloop_count:INT:=0;
	rSPEED: REAL:=2500;
	rACC:REAL:=100;
	rDCC:REAL:=100;
	r_vel_EL_temp:LREAL;
	add_vel:LREAL;
	r_vel_EL:LREAL;
	b_modify_vel: BOOL;
	b_start_adjust_vel:BOOL;
	b_start_adjust_vel_temp:BOOL;
	r_compensation_value_motor: LREAL;
	r_compensation_abs: LREAL;
	b_test_offset_start:BOOL;
	r_offset_az_old:LREAL;
	r_offset_el_old:LREAL;
(*EL  vel mode*)	
	V_LastOutput:LREAL:=0;
	V_LastSpeed:LREAL:=0;
	dIntegralSpeed:LREAL:= 0;	
	V_command_EL:LREAL:=0;
	V_command_EL_V:LREAL:=0;

	V_max_vel_motor:LREAL;
	b_start_cyclicvel: BOOL;
	b_write_el_vel: BOOL;
	m_dLastIntegral:LREAL:=0;
	m_dAUnsub1:LREAL:=0;
	m_dAUnsub2:LREAL:=0;
	m_dAEnsub1:LREAL:=0;
	m_dAEnsub2:LREAL:=0;
	m_dKa:LREAL:=0.5;
	m_dKv:LREAL:=0.1;
	
	speed1:LREAL;
	r_EL_current_when_goto_cmd:LREAL;
	T_count_goto:LREAL;
	Pos_EL_Aim:LREAL;
	r_cyclic_velocity:LREAL;
	r_cyclic_velocity_test:LREAL;
	Pos_EL_error:LREAL;
	b_step_running:BOOL:=0;
	b_step_running_az:BOOL:=0;
	b_step_running_el:BOOL:=0;
	r_step_count:DINT:=0;
	r_step_count_temp:DINT:=0;
	b_offset_running:BOOL;
	r_offset_count_temp:DINT:=0;
	r_offset_count:DINT:=0;
	r_test_offset_az:LREAL;
	r_test_offset_el:LREAL;
	r_Integral_thistime:REAL;
	r_el_offset_abs:LREAL;
END_VAR
VAR_GLOBAL RETAIN PERSISTENT
	AZ_encoder_last: LREAL;
	FI_encoder_last: LREAL;

(*	
	C1:REAL:=-0.504475;
	C2:REAL:=-0.047962;
	C3:REAL:=0.005718;
	C4:REAL:=50.64244;
	C5:REAL:=-0.003995;
	C6:REAL:=0.443004;
	C7:REAL:=0.019635;
	C8:REAL:=0;
*)	

(*	C1:LREAL:=0;
	C2:LREAL:=0;
	C3:LREAL:=0;
	C4:LREAL:=0;
	C5:LREAL:=0;
	C6:LREAL:=0;
	C7:LREAL:=0;
	C8:LREAL:=0;	
*)
	r_pos_motor3_Ini: REAL;

(*	
	P1:LREAL:=0.000000000968559949;
	P2:LREAL:=-0.000000404463748;
	P3:LREAL:=0.0000707747355;
	P4:LREAL:=-0.006745089;
	P5:LREAL:=0.3810258947;
	P6:LREAL:=-13.13945082;
	P7:LREAL:=311.5666046431;
	P8:LREAL:=4122.813236;
	P9:LREAL:=556099.6655657330;
*)
	(*P1:LREAL:=0.00000000000675664022381225;
	P2:LREAL:=-0.00000000306148315353895;
	P3:LREAL:=0.000000597917575287703;
	P4:LREAL:=-0.0000659096897179393;
	P5:LREAL:=0.00450794567760492;
	P6:LREAL:=-0.198139695223752;
	P7:LREAL:=5.43570049374671;
	P8:LREAL:=-35.3877608207139;
	P9:LREAL:=9702.49448593394;
	P10:LREAL:=422614.297996071;*)
END_VAR

// IndraMotionMlc1/Application/UserConstGlobal
VAR_GLOBAL CONSTANT
  // define all possible axis, set to maximum axis index to preserve ressources 
  // set to a maximum of 32 for the L45 and 16? for the L25
  uiMAX_AXIS_INDEX:   UINT    := INT_TO_UINT(MB_MAX_AXIS_NUMBER);
  
  // Simulation related
  gc_b_sim_on: BOOL :=1;  // True is simulation code activated. 
  // Azimuth limits
  	gc_r_limit_cw_az_sim:REAL:= 271 ;
	gc_r_limit_ccw_az_sim:REAL:= -271;
	gc_r_limit_final_cw_az_sim:REAL:= 271.2 ;
	gc_r_limit_final_ccw_az_sim:REAL:=-271.2 ;
 // Elevation Limits
	gc_r_limit_cw_el_sim:REAL:= 90.2;
	gc_r_limit_ccw_el_sim:REAL:= 14.8 ;
	gc_r_limit_final_cw_el_sim:REAL:=90.5 ;
	gc_r_limit_final_ccw_el_sim:REAL:=14.5 ;
 // Feed Indexer Limits
	gc_r_limit_cw_fi_sim:REAL:= 106;
	gc_r_limit_ccw_fi_sim:REAL:= -106;
	gc_r_limit_final_cw_fi_sim:REAL:= 106.2 ;
	gc_r_limit_final_ccw_fi_sim:REAL:= -106.2;
  
  // Time related 
  gc_UnixToSKAEpoch: LREAL := 946684768 ; //Seconds
  gc_SKAEpochMJD: LREAL := 51544; // MJD
  gc_KAPB_NTP: STRING :='10.97.64.1';
  
 (* // Position limits
  gc_r_pos_max_Az: REAL := 271;
  gc_r_pos_min_Az: REAL := -271;  
  gc_r_pos_max_El: REAL := 90.2;
  gc_r_pos_min_El: REAL := 14.8;  
  gc_r_pos_max_Fi: REAL := 106;
  gc_r_pos_min_Fi: REAL := -106;  *)

   // Position limits
  gc_r_pos_max_Az: REAL := 2710;
  gc_r_pos_min_Az: REAL := -2710;  
  gc_r_pos_max_El: REAL := 900.20;
  gc_r_pos_min_El: REAL := -14.80;  
  gc_r_pos_max_Fi: REAL := 1060;
  gc_r_pos_min_Fi: REAL := -1060;  
  
  
  // Velocity limits
   gc_r_vel_max_Az: REAL := 0.5; //3/6; //scaling RPM of Axis  Deg/s = 6* RPM 
   gc_r_vel_max_El: REAL := 0.16667;
   gc_r_vel_max_Fi: REAL := 2;
   
  // Power limiting
     gc_r_power_Kv_Az: REAL := 0.05;//0.3Deg/s/kW;
  	 gc_r_power_Kv_El: REAL := 0.016667;// 0.1;
     gc_r_power_Kv_Fi: REAL := 0.2;//1.2;
	 gc_r_power_Ka_Az: REAL := 0.055;
  	 gc_r_power_Ka_El: REAL := 0.002;
  	 gc_r_power_Ka_Fi: REAL := 0.1; 

     
   // Tracking  If the velocity is below this limit then then the dish is tracking abovethe limit it is slewing. 
   gc_r_vel_tracking_limit_Az: REAL := 1;  // Scaling
   gc_r_vel_tracking_limit_El: REAL := 0.4;
   gc_r_vel_tracking_limit_Fi: REAL := 0;
   
   // Stop Deceleration values  
  gc_r_Stop_dec_Az: REAL := 0.5; //Rad/s^2
  gc_r_Stop_dec_El: REAL := 0.5; // 28,64 deg/s^2
  gc_r_Stop_dec_Fi: REAL := 0.5;
  
   // Stop Deceleration values  
  gc_r_limit_Stop_dec_Az: REAL := 5; //Rad/s^2
  gc_r_limit_Stop_dec_El: REAL := 5; // 28,64 deg/s^2
  gc_r_limit_Stop_dec_Fi: REAL := 5;
  
  
  // Goto Acceleration Values
  gc_r_goto_acc_Az: REAL := 0.02; //Rad/s^2 
  gc_r_goto_acc_El: REAL := 0.02; // 1.14 deg/s^@
  gc_r_goto_acc_Fi: REAL := 0.2; // 11.4 deg/s^2
  
  // Feed indexer positions for bands
  gc_r_band_tolerance: REAL := 0.001; // Tolerance for being in position
  gc_r_band_optical : REAL := 0;
  gc_r_band_1 : REAL := 103.37;
  gc_r_band_2 : REAL := -99.97;
  gc_r_band_3 : REAL := -47.684;
  gc_r_band_4 : REAL := 10.444;
  gc_r_band_5a : REAL := -6.398;
  gc_r_band_5b : REAL := -30.842;
  gc_r_band_6 : REAL := -18.62;
  
  // Stow Positions
  gc_r_stow_Az: REAL :=0; 
  gc_r_stow_El: REAL :=90;
  gc_stow_horn_alarm_time: TIME := T#5S;
  gc_UPS_Stow_Az_Speed: REAL := 0.16667;
  gc_UPS_Stow_El_Speed: REAL := 0.083; 
  // AutoStow 
  gc_i_autostow_counter_max: INT := 2; 
  
  // Static off set limits
  gc_r_Xel_off_limit: REAL := 36000; // arcsec
  gc_r_El_off_limit: REAL := 36000;
	 
  // Pointing 
  gc_stack_length: INT :=12000; 
  gc_r_tilt_vel_limit_Az: REAL := 1; // deg/s	 
  gc_lr_tilt_corr_limit_Az: LREAL:= 1000; //arcseconds 
  gc_lr_tilt_corr_limit_El: LREAL:= 1000; //arcseconds 
  gc_lr_arcsec2deg: LREAL:=3600;
  gc_lr_point_corr_error_lim : LREAL := 360000; //arcseconds
	 
END_VAR

// IndraMotionMlc1/Application/UserVarGlobal
VAR_GLOBAL 
  // Axis interface: command structure: define as RETAIN, to keep the values 
  // Note: on the L40.2 control, the RETAIN memory is slower then normal VAR, so define 
  //       this structure only as RETAIN when necessary 
  //  arAxisCtrl_gb: ARRAY [1..MAX_AXIS_NUM] OF MB_AXIS_CONTROL;
	
  // Axis interface: command structure 
  arAxisCtrl_gb: ARRAY [1..uiMAX_AXIS_INDEX] OF TE_AXIS_CONTROL_TYPE01;
END_VAR

VAR_GLOBAL
//----------------------------------- Machine status variables ----------------------------	

  // Axis interface: status structure 
  arAxisStatus_gb: ARRAY [1..uiMAX_AXIS_INDEX] OF TE_AXIS_STATUS_TYPE01;

  bRemoteOn_gb  : BOOL := FALSE;  // TRUE: Internal IL visu is active 
                                  // FALSE: PlcProg is active

  
END_VAR

// IndraMotionMlc1/Application/AxisInterface/Global_AxIf_Const
{attribute 'qualified_only'}
VAR_GLOBAL CONSTANT
    // define masks for the sync operating modes 
    // e.g. IF( (INT_TO_WORD(AdminStatus._OpMode.enAck) AND MASK_MODE_WITH_FINE_ADJ) <> 0 ) THEN 
    MASK_MODE_PHASE_SHIFT   :DWORD := 16#0BC0; (* SYNC_PHASE, SYNC_CAM, SYNC_PROFILE, FLEX_PROFILE, SYNC_VEL *)
END_VAR
VAR_GLOBAL

END_VAR

// IndraMotionMlc1/Application/AxisInterface/Global_Axis_Interface
{attribute 'linkalways'}
{attribute 'analysis' := '-33'} // disable static code analysis rule 33, check of unused variable
VAR_GLOBAL
    (* Axis number for the visualization screens *)
    VisuAxisNo : INT := 1;
    
	  arAxisIdx_gb: ARRAY [1..uiMAX_AXIS_INDEX] OF UINT; // list of all axes index without gaps 
    uiNofAxis_gb: UINT; // number of axis in C-0-0484
    
END_VAR

// IndraMotionMlc1/Application/PLC_PRG
VAR_GLOBAL
		
Safety:fb_Safety;
CommandArbiter:fb_CommandArbiter;
Time_cds:fb_Time_cds;
Pointing:fb_Pointing;
Tracking:fb_Tracking;
Management:fb_Management;
Azimuth:fb_Axis;
Elevation:fb_Axis;
FeedIndexer:fb_Axis;





	
(************CommandArbiter ************)	

	Authority:STRING:='LMC';    (* the authority for DSC control now*)
	Command_Arbiter_error:BOOL;(*Command Arbiter error*)

(****************Management*******************)

	DsState:UINT;(*The Dish state 0Startup 1Standby 2Locked 3Estop 4Stowed 5Lcok&Stowed 6Activating 7Deactivating 8Standstill 9Stop 10Slew 11jog 12Track*)
	Current_FIPos:UINT;(*Current position of the FI*)
	r_operation_hour: LREAL;(*FP_C_0_0051,Operation hour counter*)
	K_gear_ratio:LREAL:=1800;// The ratio beteen the leadscrew length and elevation angle This variable needs a non-zero startup to prevent divide by zero.
	HumidDriveCab: LREAL;
	HumidPSC_Inlet: LREAL;
	HumidPSC_Outlet: LREAL;
	TempDriveCab: LREAL;
	TempEMISC_Outlet: LREAL;
	TempPSC_Inlet: LREAL;
	TempPSC_Outlet: LREAL;
	CurrentPh1: LREAL;
	CurrentPh2: LREAL;
	CurrentPh3: LREAL;
	FrequencyPh1: LREAL;
	FrequencyPh2: LREAL;
	FrequencyPh3: LREAL;
	PowerFactor: LREAL;
	VoltagePh1: LREAL;
	VoltagePh2: LREAL;
	VoltagePh3: LREAL;
	
	Pedestal_temp_1: REAL;
	Pedestal_temp_2 : REAL;
	Pedestal_temp_3 : REAL;
	
	
(********************Time**********************)	
	Source_Timesync:UINT:=2;(*Time source, 0 PTP 1 NTP 2 DSC*)
	IP_Adress_PTP:STRING;(* The PTP server adresss*)
	IP_Adress_NTP:STRING;(* The PTP server adresss*)
	//DscTime:DATE_AND_TIME;(*DSC internal time*)
	//TimeSynced:BOOL;(*The time is synced to the source*)
	
